KUKA KRL program: MyProgram_292().src

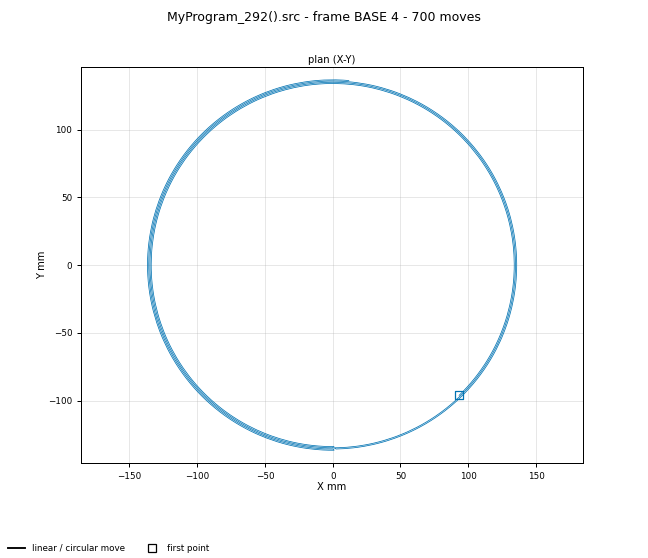
[picture p0: tool path of MyProgram_292().src in frame BASE 4, 700 of 700 moves have a stored position in this frame; points joined in program order, loops and branches not executed]
&ACCESS RVP
&REL 1
&PARAM TEMPLATE = C:\KRC\Roboter\Template\vorgabe
&PARAM EDITMASK = *
DEF MyProgram_292()
; ---- Setting reference (Base) ----
$BASE = BASE_DATA[4]

; --------------------------
; ---- Setting tool (TCP) ----
$TOOL = TOOL_DATA[3]
; --------------------------

$VEL.CP = VEL_APROX_PRINT
Startdeposition()
$VEL.CP = VEL_PRINT
LIN {X 93.2547,Y -96.1677,Z 177,A -42.5011,B 6.5222,C 0.3337,E1 6.6439,E2 494.4395} C_DIS
LIN {X 96.4506,Y -92.9625,Z 177,A -40.616,B 6.5225,C 0.3304,E1 6.6475,E2 492.5591} C_DIS
LIN {X 99.1155,Y -90.1154,Z 177,A -39.0001,B 6.5225,C 0.3277,E1 6.6506,E2 490.9482} C_DIS
LIN {X 101.7886,Y -87.0857,Z 177,A -37.2313,B 6.5228,C 0.3231,E1 6.6538,E2 489.1727} C_DIS
LIN {X 104.4652,Y -83.8557,Z 177,A -35.5009,B 6.523,C 0.3201,E1 6.6569,E2 487.4487} C_DIS
LIN {X 106.9431,Y -80.6711,Z 177,A -33.7806,B 6.5232,C 0.3162,E1 6.6598,E2 485.7275} C_DIS
LIN {X 109.619,Y -76.9961,Z 177,A -31.8796,B 6.5233,C 0.3123,E1 6.6629,E2 483.8301} C_DIS
LIN {X 112.1141,Y -73.3161,Z 177,A -30.1093,B 6.5235,C 0.3099,E1 6.6656,E2 482.0746} C_DIS
LIN {X 113.9637,Y -70.4067,Z 177,A -28.5276,B 6.5237,C 0.3044,E1 6.668,E2 480.478} C_DIS
LIN {X 115.9303,Y -67.118,Z 177,A -27.0187,B 6.5238,C 0.3025,E1 6.6701,E2 478.9839} C_DIS
LIN {X 118.1011,Y -63.2205,Z 177,A -25.0687,B 6.5241,C 0.2969,E1 6.6727,E2 477.0268} C_DIS
LIN {X 119.8057,Y -59.9271,Z 177,A -23.4735,B 6.5242,C 0.2926,E1 6.6747,E2 475.429} C_DIS
LIN {X 121.6866,Y -56.0049,Z 177,A -21.7807,B 6.5243,C 0.2906,E1 6.6767,E2 473.7555} C_DIS
LIN {X 122.9604,Y -53.1495,Z 177,A -20.5105,B 6.5244,C 0.2882,E1 6.6781,E2 472.4924} C_DIS
LIN {X 124.4377,Y -49.5951,Z 177,A -18.8101,B 6.5247,C 0.2828,E1 6.6799,E2 470.7838} C_DIS
LIN {X 125.9052,Y -45.7399,Z 177,A -17.0927,B 6.5248,C 0.2789,E1 6.6816,E2 469.0705} C_DIS
LIN {X 127.2852,Y -41.7458,Z 177,A -15.2801,B 6.5251,C 0.2738,E1 6.6832,E2 467.2556} C_DIS
LIN {X 128.7083,Y -37.1294,Z 177,A -12.2803,B 6.5259,C 0.2519,E1 6.6857,E2 464.1364} C_DIS
LIN {X 130.5683,Y -29.9352,Z 177,A -10.1949,B 6.5255,C 0.262,E1 6.6869,E2 462.1858} C_DIS
LIN {X 131.2974,Y -26.5557,Z 177,A -8.8361,B 6.5256,C 0.2599,E1 6.6877,E2 460.8406} C_DIS
LIN {X 131.8472,Y -23.6754,Z 177,A -7.5979,B 6.5258,C 0.2566,E1 6.6883,E2 459.6033} C_DIS
LIN {X 132.417,Y -20.2488,Z 177,A -6.0396,B 6.526,C 0.2511,E1 6.689,E2 458.0347} C_DIS
LIN {X 132.9133,Y -16.6972,Z 177,A -4.5118,B 6.5261,C 0.2469,E1 6.6895,E2 456.5064} C_DIS
LIN {X 133.3452,Y -12.7791,Z 177,A -2.9752,B 6.5262,C 0.2446,E1 6.69,E2 454.9869} C_DIS
LIN {X 133.6654,Y -8.842,Z 177,A -1.0029,B 6.5266,C 0.2349,E1 6.6904,E2 452.978} C_DIS
LIN {X 133.8408,Y -5.5702,Z 177,A -0.0788,B 6.5264,C 0.2391,E1 6.6904,E2 452.112} C_DIS
LIN {X 133.9241,Y -3.0185,Z 177,A 1.1002,B 6.5266,C 0.2345,E1 6.6906,E2 450.9214} C_DIS
LIN {X 133.9546,Y 0.822,Z 177,A 2.8788,B 6.5268,C 0.2274,E1 6.6906,E2 449.1246} C_DIS
LIN {X 133.879,Y 4.576,Z 177,A 4.2711,B 6.5268,C 0.2265,E1 6.6905,E2 447.7575} C_DIS
LIN {X 133.7434,Y 7.5752,Z 177,A 5.4943,B 6.527,C 0.2239,E1 6.6903,E2 446.5409} C_DIS
LIN {X 133.4661,Y 11.4487,Z 177,A 7.1189,B 6.527,C 0.2198,E1 6.6899,E2 444.9194} C_DIS
LIN {X 133.2196,Y 14.0308,Z 177,A 8.1651,B 6.5272,C 0.2177,E1 6.6897,E2 443.8802} C_DIS
LIN {X 132.9288,Y 16.5728,Z 177,A 9.3123,B 6.5272,C 0.2137,E1 6.6893,E2 442.7257} C_DIS
LIN {X 132.5516,Y 19.3507,Z 177,A 10.6317,B 6.5275,C 0.2082,E1 6.6887,E2 441.3905} C_DIS
LIN {X 131.8477,Y 23.6726,Z 177,A 12.355,B 6.5275,C 0.2055,E1 6.6879,E2 439.6844} C_DIS
LIN {X 131.2568,Y 26.7556,Z 177,A 13.6501,B 6.5277,C 0.2026,E1 6.6872,E2 438.3942} C_DIS
LIN {X 130.5423,Y 30.0492,Z 177,A 15.1238,B 6.5277,C 0.198,E1 6.6863,E2 436.9154} C_DIS
LIN {X 129.489,Y 34.3048,Z 177,A 16.9836,B 6.5279,C 0.1931,E1 6.685,E2 435.0563} C_DIS
LIN {X 128.2952,Y 38.5354,Z 177,A 19.333,B 6.5283,C 0.1799,E1 6.6831,E2 432.6477} C_DIS
LIN {X 126.8174,Y 43.1518,Z 177,A 20.7515,B 6.5282,C 0.1854,E1 6.682,E2 431.3088} C_DIS
LIN {X 124.899,Y 48.419,Z 177,A 23.6983,B 6.5286,C 0.1697,E1 6.679,E2 428.2928} C_DIS
LIN {X 123.0953,Y 52.8375,Z 177,A 24.9449,B 6.5284,C 0.1778,E1 6.6777,E2 427.1429} C_DIS
LIN {X 121.1405,Y 57.1795,Z 177,A 27.275,B 6.5286,C 0.1676,E1 6.675,E2 424.7758} C_DIS
LIN {X 119.2439,Y 61.0336,Z 177,A 28.926,B 6.5286,C 0.166,E1 6.6729,E2 423.1466} C_DIS
LIN {X 117.5054,Y 64.3209,Z 177,A 30.6108,B 6.5288,C 0.1604,E1 6.6707,E2 421.4496} C_DIS
LIN {X 115.2166,Y 68.3366,Z 177,A 32.5475,B 6.5289,C 0.1562,E1 6.668,E2 419.517} C_DIS
LIN {X 112.8881,Y 72.1176,Z 177,A 34.404,B 6.529,C 0.1523,E1 6.6652,E2 417.6649} C_DIS
LIN {X 110.2862,Y 76.0374,Z 177,A 36.2624,B 6.529,C 0.1501,E1 6.6623,E2 415.8244} C_DIS
LIN {X 107.7865,Y 79.5413,Z 177,A 38.1742,B 6.5292,C 0.1447,E1 6.6592,E2 413.9033} C_DIS
LIN {X 101.9515,Y 86.8941,Z 177,A 42.0062,B 6.5293,C 0.1388,E1 6.6525,E2 410.0924} C_DIS
LIN {X 99.4872,Y 89.7057,Z 177,A 43.7299,B 6.5294,C 0.1333,E1 6.6493,E2 408.353} C_DIS
LIN {X 96.1576,Y 93.2651,Z 177,A 45.6306,B 6.5294,C 0.132,E1 6.6457,E2 406.4741} C_DIS
LIN {X 93.4408,Y 95.9875,Z 177,A 47.3771,B 6.5295,C 0.127,E1 6.6422,E2 404.7149} C_DIS
LIN {X 90.2793,Y 98.9668,Z 177,A 49.225,B 6.5296,C 0.1236,E1 6.6384,E2 402.8678} C_DIS
LIN {X 87.6848,Y 101.2726,Z 177,A 50.6916,B 6.5296,C 0.1211,E1 6.6353,E2 401.4032} C_DIS
LIN {X 84.3245,Y 104.0871,Z 177,A 52.5309,B 6.5297,C 0.1182,E1 6.6313,E2 399.5678} C_DIS
LIN {X 80.8508,Y 106.8075,Z 177,A 54.3017,B 6.5297,C 0.1168,E1 6.6275,E2 397.8109} C_DIS
LIN {X 77.4949,Y 109.267,Z 177,A 56.7417,B 6.53,C 0.1034,E1 6.6217,E2 395.2904} C_DIS
LIN {X 72.9543,Y 112.3491,Z 177,A 58.2306,B 6.5298,C 0.1131,E1 6.6185,E2 393.9056} C_DIS
LIN {X 70.2551,Y 114.0567,Z 177,A 59.8013,B 6.5298,C 0.1079,E1 6.6147,E2 392.3102} C_DIS
LIN {X 67.1093,Y 115.9354,Z 177,A 61.3332,B 6.5299,C 0.1061,E1 6.611,E2 390.7826} C_DIS
LIN {X 63.6933,Y 117.8471,Z 177,A 63.0269,B 6.5299,C 0.1035,E1 6.6069,E2 389.0865} C_DIS
LIN {X 59.6278,Y 119.9533,Z 177,A 64.965,B 6.5299,C 0.1013,E1 6.602,E2 387.1509} C_DIS
LIN {X 55.7819,Y 121.7897,Z 177,A 66.6368,B 6.5299,C 0.1013,E1 6.5979,E2 385.4974} C_DIS
LIN {X 52.4854,Y 123.2475,Z 177,A 68.1681,B 6.53,C 0.0997,E1 6.5939,E2 383.9676} C_DIS
LIN {X 49.6492,Y 124.4159,Z 177,A 69.4709,B 6.53,C 0.0984,E1 6.5906,E2 382.666} C_DIS
LIN {X 45.9682,Y 125.8229,Z 177,A 71.4893,B 6.5301,C 0.0918,E1 6.5852,E2 380.6076} C_DIS
LIN {X 42.6946,Y 126.9704,Z 177,A 72.6051,B 6.5301,C 0.0958,E1 6.5824,E2 379.5365} C_DIS
LIN {X 35.9258,Y 129.0486,Z 177,A 75.9572,B 6.5301,C 0.0886,E1 6.5733,E2 376.1461} C_DIS
LIN {X 32.5628,Y 129.9385,Z 177,A 77.0114,B 6.5301,C 0.0938,E1 6.5706,E2 375.1444} C_DIS
LIN {X 29.6776,Y 130.6272,Z 177,A 78.365,B 6.5301,C 0.0917,E1 6.5669,E2 373.781} C_DIS
LIN {X 26.4894,Y 131.3109,Z 177,A 79.7722,B 6.5301,C 0.0907,E1 6.563,E2 372.3726} C_DIS
LIN {X 22.8852,Y 131.9886,Z 177,A 81.2873,B 6.5301,C 0.0907,E1 6.5589,E2 370.8645} C_DIS
LIN {X 19.5056,Y 132.5295,Z 177,A 82.849,B 6.5301,C 0.0886,E1 6.5545,E2 369.2915} C_DIS
LIN {X 15.2294,Y 133.0891,Z 177,A 84.594,B 6.5301,C 0.0894,E1 6.5497,E2 367.5591} C_DIS
LIN {X 11.0703,Y 133.4981,Z 177,A 86.315,B 6.5301,C 0.0898,E1 6.545,E2 365.8467} C_DIS
LIN {X 8.5569,Y 133.683,Z 177,A 87.5726,B 6.5302,C 0.0871,E1 6.5414,E2 364.568} C_DIS
LIN {X 4.6226,Y 133.8778,Z 177,A 89.1069,B 6.5302,C 0.0889,E1 6.5372,E2 363.0525} C_DIS
LIN {X 1.7234,Y 133.9461,Z 177,A 90.568,B 6.5302,C 0.0858,E1 6.533,E2 361.5654} C_DIS
LIN {X -2.809,Y 133.9281,Z 177,A 92.3744,B 6.5302,C 0.0876,E1 6.528,E2 359.7758} C_DIS
LIN {X -6.0372,Y 133.8219,Z 177,A 93.7882,B 6.5302,C 0.0873,E1 6.524,E2 358.3588} C_DIS
LIN {X -9.8651,Y 133.5924,Z 177,A 95.4536,B 6.5302,C 0.0873,E1 6.5194,E2 356.6912} C_DIS
LIN {X -14.4166,Y 133.1781,Z 177,A 97.3355,B 6.5302,C 0.0888,E1 6.5142,E2 354.819} C_DIS
LIN {X -17.6905,Y 132.7831,Z 177,A 98.7772,B 6.5302,C 0.0888,E1 6.5102,E2 353.3743} C_DIS
LIN {X -21.9534,Y 132.1449,Z 177,A 100.6192,B 6.5302,C 0.0897,E1 6.5051,E2 351.5336} C_DIS
LIN {X -25.4976,Y 131.5074,Z 177,A 102.0736,B 6.5302,C 0.0916,E1 6.5012,E2 350.0903} C_DIS
LIN {X -28.3851,Y 130.9141,Z 177,A 103.3903,B 6.5302,C 0.0916,E1 6.4975,E2 348.7677} C_DIS
LIN {X -32.2156,Y 130.0266,Z 177,A 105.0573,B 6.5302,C 0.0929,E1 6.493,E2 347.1036} C_DIS
LIN {X -34.716,Y 129.3794,Z 177,A 106.2071,B 6.5302,C 0.0931,E1 6.4899,E2 345.949} C_DIS
LIN {X -40.4025,Y 127.7182,Z 177,A 108.5712,B 6.5301,C 0.0973,E1 6.4836,E2 343.607} C_DIS
LIN {X -44.6966,Y 126.2813,Z 177,A 111.3947,B 6.5301,C 0.0878,E1 6.4759,E2 340.6783} C_DIS
LIN {X -49.5868,Y 124.441,Z 177,A 112.8347,B 6.5301,C 0.1001,E1 6.4724,E2 339.3355} C_DIS
LIN {X -51.7604,Y 123.5517,Z 177,A 114.0213,B 6.5301,C 0.0989,E1 6.4693,E2 338.1279} C_DIS
LIN {X -55.3587,Y 121.9839,Z 177,A 115.6589,B 6.53,C 0.1014,E1 6.4651,E2 336.4965} C_DIS
LIN {X -58.1429,Y 120.6802,Z 177,A 117.1082,B 6.53,C 0.1014,E1 6.4614,E2 335.032} C_DIS
LIN {X -61.7821,Y 118.8587,Z 177,A 119.1939,B 6.53,C 0.0994,E1 6.4562,E2 332.9061} C_DIS
LIN {X -65.3727,Y 116.9237,Z 177,A 120.3017,B 6.5299,C 0.1096,E1 6.4537,E2 331.8762} C_DIS
LIN {X -67.9903,Y 115.421,Z 177,A 121.9186,B 6.5299,C 0.1075,E1 6.4496,E2 330.2213} C_DIS
LIN {X -71.3651,Y 113.3653,Z 177,A 123.619,B 6.5299,C 0.1099,E1 6.4456,E2 328.5211} C_DIS
LIN {X -76.8897,Y 109.694,Z 177,A 126.2273,B 6.5297,C 0.1171,E1 6.4397,E2 325.9426} C_DIS
LIN {X -79.3379,Y 107.9359,Z 177,A 127.799,B 6.5297,C 0.1159,E1 6.436,E2 324.3381} C_DIS
LIN {X -82.8055,Y 105.2991,Z 177,A 129.6731,B 6.5297,C 0.1191,E1 6.4319,E2 322.4643} C_DIS
LIN {X -86.1951,Y 102.5431,Z 177,A 131.5799,B 6.5297,C 0.122,E1 6.4278,E2 320.5545} C_DIS
LIN {X -89.4519,Y 99.7147,Z 177,A 133.4568,B 6.5296,C 0.1252,E1 6.4238,E2 318.6753} C_DIS
LIN {X -92.8056,Y 96.6017,Z 177,A 135.4367,B 6.5296,C 0.1287,E1 6.4198,E2 316.6944} C_DIS
LIN {X -95.7212,Y 93.7129,Z 177,A 137.2067,B 6.5294,C 0.1321,E1 6.4163,E2 314.9243} C_DIS
LIN {X -98.7785,Y 90.4849,Z 177,A 139.1704,B 6.5294,C 0.1354,E1 6.4126,E2 312.9547} C_DIS
LIN {X -101.7402,Y 87.142,Z 177,A 141.1279,B 6.5294,C 0.139,E1 6.409,E2 310.9933} C_DIS
LIN {X -104.577,Y 83.7165,Z 177,A 143.05,B 6.5292,C 0.143,E1 6.4056,E2 309.0706} C_DIS
LIN {X -107.1431,Y 80.4061,Z 177,A 144.7491,B 6.5292,C 0.1482,E1 6.4027,E2 307.3842} C_DIS
LIN {X -109.243,Y 77.5291,Z 177,A 146.4559,B 6.5291,C 0.1497,E1 6.3999,E2 305.6568} C_DIS
LIN {X -112.9435,Y 72.0311,Z 177,A 149.2423,B 6.5289,C 0.157,E1 6.3956,E2 302.8788} C_DIS
LIN {X -115.0741,Y 68.5756,Z 177,A 151.0676,B 6.5289,C 0.1603,E1 6.393,E2 301.0444} C_DIS
LIN {X -116.8004,Y 65.5922,Z 177,A 152.5887,B 6.5287,C 0.1634,E1 6.3909,E2 299.519} C_DIS
LIN {X -118.933,Y 61.6406,Z 177,A 154.4238,B 6.5286,C 0.1692,E1 6.3885,E2 297.6959} C_DIS
LIN {X -120.4075,Y 58.7071,Z 177,A 155.9944,B 6.5286,C 0.171,E1 6.3865,E2 296.1066} C_DIS
LIN {X -123.0186,Y 53.015,Z 177,A 158.6392,B 6.5284,C 0.1784,E1 6.3835,E2 293.4683} C_DIS
LIN {X -124.3654,Y 49.7743,Z 177,A 160.1661,B 6.5283,C 0.1821,E1 6.3819,E2 291.9397} C_DIS
LIN {X -125.8482,Y 45.8979,Z 177,A 161.8282,B 6.5281,C 0.1881,E1 6.3803,E2 290.2929} C_DIS
LIN {X -126.6044,Y 43.7664,Z 177,A 163.0259,B 6.5281,C 0.1883,E1 6.3792,E2 289.0681} C_DIS
LIN {X -127.7431,Y 40.3247,Z 177,A 164.4677,B 6.5279,C 0.1937,E1 6.3779,E2 287.641} C_DIS
LIN {X -128.7727,Y 36.9097,Z 177,A 166.0775,B 6.5279,C 0.197,E1 6.3767,E2 286.0223} C_DIS
LIN {X -129.7111,Y 33.4588,Z 177,A 167.5354,B 6.5277,C 0.202,E1 6.3756,E2 284.5745} C_DIS
LIN {X -130.611,Y 29.7484,Z 177,A 169.3185,B 6.5276,C 0.2049,E1 6.3745,E2 282.7746} C_DIS
LIN {X -131.3492,Y 26.3015,Z 177,A 171.0086,B 6.5276,C 0.2072,E1 6.3735,E2 281.0637} C_DIS
LIN {X -132.1843,Y 21.7173,Z 177,A 172.9941,B 6.5273,C 0.2129,E1 6.3725,E2 279.0809} C_DIS
LIN {X -132.7482,Y 17.957,Z 177,A 174.509,B 6.5271,C 0.2188,E1 6.3719,E2 277.581} C_DIS
LIN {X -133.1057,Y 15.0892,Z 177,A 175.8069,B 6.5271,C 0.2216,E1 6.3715,E2 276.2767} C_DIS
LIN {X -133.4911,Y 11.1532,Z 177,A 177.5894,B 6.5269,C 0.2255,E1 6.3711,E2 274.4844} C_DIS
LIN {X -133.771,Y 7.049,Z 177,A 179.4151,B 6.5268,C 0.2298,E1 6.3708,E2 272.6522} C_DIS
LIN {X -133.9146,Y 3.3582,Z 177,A -179.067,B 6.5266,C 0.235,E1 6.3706,E2 271.1432} C_DIS
LIN {X -133.9568,Y 0.5032,Z 177,A -177.7907,B 6.5265,C 0.2379,E1 6.3706,E2 269.8612} C_DIS
LIN {X -133.9184,Y -3.2227,Z 177,A -176.0516,B 6.5264,C 0.2409,E1 6.3706,E2 268.1055} C_DIS
LIN {X -133.7767,Y -6.9356,Z 177,A -174.5652,B 6.5261,C 0.2465,E1 6.3709,E2 266.6329} C_DIS
LIN {X -133.5934,Y -9.8526,Z 177,A -173.2029,B 6.5261,C 0.2489,E1 6.3711,E2 265.2578} C_DIS
LIN {X -133.2061,Y -14.1561,Z 177,A -171.2366,B 6.5259,C 0.2528,E1 6.3717,E2 263.2785} C_DIS
LIN {X -132.6335,Y -18.7776,Z 177,A -169.2218,B 6.5257,C 0.2582,E1 6.3724,E2 261.2624} C_DIS
LIN {X -132.1135,Y -22.1417,Z 177,A -167.8158,B 6.5255,C 0.2629,E1 6.373,E2 259.8636} C_DIS
LIN {X -131.4967,Y -25.5535,Z 177,A -166.373,B 6.5253,C 0.2675,E1 6.3738,E2 258.4268} C_DIS
LIN {X -130.815,Y -28.8441,Z 177,A -164.5422,B 6.5253,C 0.2672,E1 6.3749,E2 256.5485} C_DIS
LIN {X -128.9504,Y -36.2767,Z 177,A -161.3851,B 6.5249,C 0.2775,E1 6.3771,E2 253.4086} C_DIS
LIN {X -127.969,Y -39.6012,Z 177,A -159.8428,B 6.5248,C 0.2809,E1 6.3784,E2 251.8598} C_DIS
LIN {X -126.8559,Y -43.0385,Z 177,A -158.4005,B 6.5245,C 0.2862,E1 6.3796,E2 250.4313} C_DIS
LIN {X -125.6963,Y -46.3153,Z 177,A -156.9142,B 6.5244,C 0.2902,E1 6.381,E2 248.9459} C_DIS
LIN {X -124.7138,Y -48.8954,Z 177,A -155.6899,B 6.5242,C 0.2928,E1 6.3823,E2 247.7169} C_DIS
LIN {X -123.2773,Y -52.4166,Z 177,A -154.0105,B 6.5241,C 0.2965,E1 6.3841,E2 246.032} C_DIS
LIN {X -121.9963,Y -55.331,Z 177,A -152.618,B 6.5239,C 0.2996,E1 6.3857,E2 244.6364} C_DIS
LIN {X -120.0449,Y -59.4422,Z 177,A -150.5894,B 6.5237,C 0.3036,E1 6.3881,E2 242.5986} C_DIS
LIN {X -118.4513,Y -62.5579,Z 177,A -148.1294,B 6.5241,C 0.2964,E1 6.3915,E2 240.0192} C_DIS
LIN {X -115.1617,Y -68.4287,Z 177,A -146.0824,B 6.5233,C 0.313,E1 6.3942,E2 238.0777} C_DIS
LIN {X -112.864,Y -72.1553,Z 177,A -144.1833,B 6.5231,C 0.3171,E1 6.3971,E2 236.1762} C_DIS
LIN {X -110.4263,Y -75.8333,Z 177,A -142.2092,B 6.5229,C 0.3205,E1 6.4002,E2 234.1921} C_DIS
LIN {X -107.7448,Y -79.598,Z 177,A -140.4774,B 6.5226,C 0.3278,E1 6.4029,E2 232.4915} C_DIS
LIN {X -106.0986,Y -81.7795,Z 177,A -138.87,B 6.5227,C 0.3253,E1 6.4058,E2 230.8299} C_DIS
LIN {X -103.506,Y -85.0369,Z 177,A -137.1986,B 6.5225,C 0.3304,E1 6.4087,E2 229.1728} C_DIS
LIN {X -100.6101,Y -88.4444,Z 177,A -135.2447,B 6.5223,C 0.3339,E1 6.4123,E2 227.2144} C_DIS
LIN {X -98.2184,Y -91.0927,Z 177,A -133.758,B 6.5221,C 0.3375,E1 6.4151,E2 225.733} C_DIS
LIN {X -95.549,Y -93.8885,Z 177,A -132.0971,B 6.5219,C 0.3407,E1 6.4183,E2 224.0716} C_DIS
LIN {X -92.7691,Y -96.6366,Z 177,A -130.3072,B 6.5219,C 0.3425,E1 6.4219,E2 222.2674} C_DIS
LIN {X -89.5256,Y -99.6487,Z 177,A -128.4052,B 6.5217,C 0.3459,E1 6.4258,E2 220.3647} C_DIS
LIN {X -86.0607,Y -102.6558,Z 177,A -126.4402,B 6.5215,C 0.3494,E1 6.43,E2 218.3997} C_DIS
LIN {X -82.3757,Y -105.6364,Z 177,A -124.476,B 6.5212,C 0.3536,E1 6.4343,E2 216.4437} C_DIS
LIN {X -79.5559,Y -107.7757,Z 177,A -122.4217,B 6.5215,C 0.3493,E1 6.4391,E2 214.3217} C_DIS
LIN {X -75.9885,Y -110.3198,Z 177,A -121.1933,B 6.5209,C 0.3603,E1 6.4417,E2 213.1745} C_DIS
LIN {X -73.3161,Y -112.1141,Z 177,A -119.5903,B 6.5209,C 0.3595,E1 6.4455,E2 211.5434} C_DIS
LIN {X -69.7205,Y -114.3847,Z 177,A -117.679,B 6.5209,C 0.3609,E1 6.45,E2 209.6205} C_DIS
LIN {X -66.3323,Y -116.3817,Z 177,A -116.0487,B 6.5207,C 0.3638,E1 6.454,E2 207.9967} C_DIS
LIN {X -62.6117,Y -118.4231,Z 177,A -114.1444,B 6.5207,C 0.3649,E1 6.4587,E2 206.0811} C_DIS
LIN {X -58.7482,Y -120.3873,Z 177,A -112.4268,B 6.5204,C 0.3689,E1 6.4629,E2 204.3806} C_DIS
LIN {X -56.2707,Y -121.5637,Z 177,A -111.2394,B 6.5204,C 0.37,E1 6.4659,E2 203.1912} C_DIS
LIN {X -52.6057,Y -123.1955,Z 177,A -109.4964,B 6.5203,C 0.3714,E1 6.4704,E2 201.4448} C_DIS
LIN {X -50.1212,Y -124.2256,Z 177,A -108.3301,B 6.5203,C 0.3723,E1 6.4734,E2 200.2762} C_DIS
LIN {X -45.5141,Y -125.9866,Z 177,A -106.3135,B 6.52,C 0.3755,E1 6.4787,E2 198.271} C_DIS
LIN {X -39.0025,Y -128.1523,Z 177,A -102.9244,B 6.5202,C 0.3716,E1 6.4878,E2 194.8242} C_DIS
LIN {X -35.6668,Y -129.121,Z 177,A -101.8519,B 6.5199,C 0.3782,E1 6.4906,E2 193.8036} C_DIS
LIN {X -32.7186,Y -129.8989,Z 177,A -100.476,B 6.5199,C 0.378,E1 6.4943,E2 192.4183} C_DIS
LIN {X -29.396,Y -130.6915,Z 177,A -98.9977,B 6.5199,C 0.3786,E1 6.4984,E2 190.9375} C_DIS
LIN {X -26.0141,Y -131.4077,Z 177,A -97.3468,B 6.5199,C 0.3769,E1 6.5029,E2 189.2645} C_DIS
LIN {X -21.9874,Y -132.1392,Z 177,A -95.6946,B 6.5199,C 0.3789,E1 6.5074,E2 187.624} C_DIS
LIN {X -18.1984,Y -132.7163,Z 177,A -94.1313,B 6.5197,C 0.3804,E1 6.5117,E2 186.0698} C_DIS
LIN {X -14.1879,Y -133.2027,Z 177,A -92.2621,B 6.5198,C 0.3788,E1 6.517,E2 184.182} C_DIS
LIN {X -10.5884,Y -133.5388,Z 177,A -90.8598,B 6.5198,C 0.381,E1 6.5208,E2 182.7973} C_DIS
LIN {X -6.8406,Y -133.7815,Z 177,A -89.1543,B 6.5198,C 0.3797,E1 6.5256,E2 181.0787} C_DIS
LIN {X -2.7749,Y -133.9286,Z 177,A -87.4107,B 6.5198,C 0.3795,E1 6.5305,E2 179.3339} C_DIS
LIN {X 0.9684,Y -133.9528,Z 177,A -86.2768,B 6.5194,C 0.3861,E1 6.5335,E2 178.258} C_DIS
Enddeposition()
LIN {X 0.9684,Y -133.9528,Z 177,A -86.2768,B 6.5194,C 0.3861,E1 6.5335,E2 178.258} C_DIS
Startdeposition()
$VEL.CP = VEL_PRINT
LIN {X -0.1253,Y -134.8623,Z 177,A -87.3645,B 6.5183,C 0.3988,E1 6.5298,E2 179.4573} C_DIS
LIN {X -3.8984,Y -134.8047,Z 177,A -88.8873,B 6.5183,C 0.3977,E1 6.5256,E2 180.9707} C_DIS
LIN {X -7.4524,Y -134.6566,Z 177,A -90.1989,B 6.5186,C 0.3949,E1 6.522,E2 182.258} C_DIS
LIN {X -11.2849,Y -134.388,Z 177,A -91.6976,B 6.5186,C 0.3928,E1 6.5179,E2 183.7406} C_DIS
LIN {X -18.9352,Y -133.525,Z 177,A -94.8815,B 6.5188,C 0.3909,E1 6.5091,E2 186.9148} C_DIS
LIN {X -22.0313,Y -133.0492,Z 177,A -96.3146,B 6.5188,C 0.3919,E1 6.5051,E2 188.3612} C_DIS
LIN {X -25.6748,Y -132.3947,Z 177,A -98.002,B 6.5187,C 0.3928,E1 6.5004,E2 190.0635} C_DIS
LIN {X -29.7309,Y -131.5431,Z 177,A -99.6989,B 6.5187,C 0.3911,E1 6.4958,E2 191.7529} C_DIS
LIN {X -32.9181,Y -130.7818,Z 177,A -101.0206,B 6.5189,C 0.3893,E1 6.4922,E2 193.066} C_DIS
LIN {X -36.0986,Y -129.9397,Z 177,A -102.3929,B 6.5189,C 0.3881,E1 6.4886,E2 194.4356} C_DIS
LIN {X -38.4704,Y -129.2586,Z 177,A -103.5047,B 6.5189,C 0.3882,E1 6.4855,E2 195.5556} C_DIS
LIN {X -44.5061,Y -127.3056,Z 177,A -106.2679,B 6.519,C 0.387,E1 6.4782,E2 198.3279} C_DIS
LIN {X -48.2453,Y -125.9373,Z 177,A -107.8626,B 6.5192,C 0.3842,E1 6.4741,E2 199.9106} C_DIS
LIN {X -51.6391,Y -124.5828,Z 177,A -109.5405,B 6.5192,C 0.3844,E1 6.4697,E2 201.6044} C_DIS
LIN {X -54.7986,Y -123.2256,Z 177,A -110.9861,B 6.5192,C 0.3827,E1 6.466,E2 203.0483} C_DIS
LIN {X -57.9363,Y -121.7816,Z 177,A -112.5318,B 6.5193,C 0.3821,E1 6.462,E2 204.6039} C_DIS
LIN {X -61.1039,Y -120.2234,Z 177,A -113.952,B 6.5195,C 0.3793,E1 6.4585,E2 206.0142} C_DIS
LIN {X -64.3645,Y -118.5122,Z 177,A -115.6527,B 6.5195,C 0.3791,E1 6.4543,E2 207.7321} C_DIS
LIN {X -68.2558,Y -116.3144,Z 177,A -117.5419,B 6.5196,C 0.3764,E1 6.4497,E2 209.6201} C_DIS
LIN {X -72.0083,Y -114.0293,Z 177,A -119.4512,B 6.5198,C 0.3743,E1 6.4452,E2 211.5346} C_DIS
LIN {X -75.8494,Y -111.5116,Z 177,A -121.169,B 6.5201,C 0.3685,E1 6.4412,E2 213.2232} C_DIS
LIN {X -79.536,Y -108.9124,Z 177,A -123.5047,B 6.52,C 0.3707,E1 6.4358,E2 215.611} C_DIS
LIN {X -83.7433,Y -105.7116,Z 177,A -125.6786,B 6.5202,C 0.366,E1 6.431,E2 217.7756} C_DIS
LIN {X -87.4973,Y -102.6262,Z 177,A -127.7456,B 6.5204,C 0.3624,E1 6.4266,E2 219.8426} C_DIS
LIN {X -90.8719,Y -99.6509,Z 177,A -129.6895,B 6.5206,C 0.3593,E1 6.4226,E2 221.7902} C_DIS
LIN {X -94.0855,Y -96.6227,Z 177,A -131.6015,B 6.5208,C 0.3562,E1 6.4187,E2 223.7062} C_DIS
LIN {X -97.0469,Y -93.6474,Z 177,A -133.3214,B 6.521,C 0.3519,E1 6.4153,E2 225.4178} C_DIS
LIN {X -99.005,Y -91.5755,Z 177,A -134.8011,B 6.521,C 0.3526,E1 6.4125,E2 226.9304} C_DIS
LIN {X -102.4643,Y -87.6877,Z 177,A -136.9033,B 6.5213,C 0.3467,E1 6.4086,E2 229.0185} C_DIS
LIN {X -105.6782,Y -83.7859,Z 177,A -139.5499,B 6.5213,C 0.3479,E1 6.4039,E2 231.7258} C_DIS
LIN {X -108.5854,Y -79.982,Z 177,A -140.9031,B 6.5219,C 0.3355,E1 6.4018,E2 232.9943} C_DIS
LIN {X -110.2852,Y -77.6213,Z 177,A -142.8241,B 6.5216,C 0.3405,E1 6.3986,E2 234.9993} C_DIS
LIN {X -112.8316,Y -73.8718,Z 177,A -144.294,B 6.5221,C 0.3308,E1 6.3964,E2 236.4124} C_DIS
LIN {X -115.0267,Y -70.4043,Z 177,A -146.0764,B 6.5223,C 0.3271,E1 6.3937,E2 238.1988} C_DIS
LIN {X -118.0456,Y -65.216,Z 177,A -149.1035,B 6.5223,C 0.3262,E1 6.3895,E2 241.2833} C_DIS
LIN {X -119.9785,Y -61.5849,Z 177,A -150.4338,B 6.5228,C 0.3172,E1 6.3879,E2 242.5615} C_DIS
LIN {X -121.4846,Y -58.5582,Z 177,A -152.0401,B 6.5228,C 0.3154,E1 6.3859,E2 244.1879} C_DIS
LIN {X -123.5502,Y -54.0652,Z 177,A -154.1328,B 6.5231,C 0.3099,E1 6.3835,E2 246.2784} C_DIS
LIN {X -125.0131,Y -50.5878,Z 177,A -155.6432,B 6.5234,C 0.3047,E1 6.3819,E2 247.7766} C_DIS
LIN {X -126.9204,Y -45.5918,Z 177,A -157.9289,B 6.5236,C 0.2988,E1 6.3796,E2 250.0626} C_DIS
LIN {X -127.8897,Y -42.7977,Z 177,A -159.2859,B 6.5237,C 0.2966,E1 6.3784,E2 251.4312} C_DIS
LIN {X -128.8416,Y -39.8419,Z 177,A -161.061,B 6.5237,C 0.298,E1 6.3769,E2 253.2611} C_DIS
LIN {X -129.9875,Y -35.9278,Z 177,A -161.9376,B 6.5243,C 0.2839,E1 6.3763,E2 254.0317} C_DIS
LIN {X -131.4598,Y -30.0952,Z 177,A -164.9497,B 6.5243,C 0.2819,E1 6.3742,E2 257.0984} C_DIS
LIN {X -132.1694,Y -26.808,Z 177,A -166.468,B 6.5245,C 0.2788,E1 6.3733,E2 258.6267} C_DIS
LIN {X -132.9616,Y -22.5559,Z 177,A -168.3487,B 6.5247,C 0.2741,E1 6.3724,E2 260.5113} C_DIS
LIN {X -133.576,Y -18.5784,Z 177,A -170.1782,B 6.5249,C 0.2706,E1 6.3717,E2 262.3542} C_DIS
LIN {X -134.089,Y -14.4084,Z 177,A -171.8696,B 6.5251,C 0.2645,E1 6.3711,E2 264.0329} C_DIS
LIN {X -134.3979,Y -11.1675,Z 177,A -173.3627,B 6.5252,C 0.2618,E1 6.3707,E2 265.5383} C_DIS
LIN {X -134.6773,Y -7.041,Z 177,A -175.1502,B 6.5254,C 0.2571,E1 6.3704,E2 267.3281} C_DIS
LIN {X -134.8247,Y -3.1804,Z 177,A -176.7847,B 6.5256,C 0.2523,E1 6.3703,E2 268.9605} C_DIS
LIN {X -134.8643,Y 0.1004,Z 177,A -178.3851,B 6.5256,C 0.2506,E1 6.3703,E2 270.585} C_DIS
LIN {X -134.7871,Y 4.5235,Z 177,A 179.7274,B 6.5259,C 0.2453,E1 6.3704,E2 272.4719} C_DIS
LIN {X -134.5783,Y 8.7378,Z 177,A 177.9383,B 6.5261,C 0.2401,E1 6.3707,E2 274.259} C_DIS
LIN {X -134.2499,Y 12.8226,Z 177,A 176.1701,B 6.5262,C 0.2354,E1 6.3711,E2 276.029} C_DIS
LIN {X -133.7905,Y 16.9664,Z 177,A 174.374,B 6.5264,C 0.2306,E1 6.3717,E2 277.8266} C_DIS
LIN {X -133.2476,Y 20.7974,Z 177,A 172.7283,B 6.5266,C 0.226,E1 6.3724,E2 279.471} C_DIS
LIN {X -132.5311,Y 24.9614,Z 177,A 170.8601,B 6.5267,C 0.2217,E1 6.3733,E2 281.3465} C_DIS
LIN {X -131.7898,Y 28.616,Z 177,A 169.2781,B 6.5269,C 0.2172,E1 6.3742,E2 282.9269} C_DIS
LIN {X -130.963,Y 32.1943,Z 177,A 167.7151,B 6.5269,C 0.2129,E1 6.3752,E2 284.4888} C_DIS
LIN {X -130.1284,Y 35.4184,Z 177,A 166.1433,B 6.5271,C 0.2107,E1 6.3764,E2 286.0784} C_DIS
LIN {X -129.1206,Y 38.9301,Z 177,A 164.6908,B 6.5272,C 0.2053,E1 6.3775,E2 287.5174} C_DIS
LIN {X -128.1439,Y 42.0344,Z 177,A 163.3201,B 6.5274,C 0.2014,E1 6.3787,E2 288.8854} C_DIS
LIN {X -127.4483,Y 44.0943,Z 177,A 161.8531,B 6.5273,C 0.2047,E1 6.3801,E2 290.4168} C_DIS
LIN {X -126.0121,Y 48.0514,Z 177,A 160.3252,B 6.5275,C 0.1971,E1 6.3816,E2 291.912} C_DIS
LIN {X -124.5495,Y 51.7188,Z 177,A 158.7781,B 6.5277,C 0.1913,E1 6.3832,E2 293.4418} C_DIS
LIN {X -123.1137,Y 55.0487,Z 177,A 157.0108,B 6.5277,C 0.1897,E1 6.3852,E2 295.2349} C_DIS
LIN {X -121.2164,Y 59.1126,Z 177,A 154.7498,B 6.5277,C 0.1886,E1 6.388,E2 297.5368} C_DIS
LIN {X -119.3107,Y 62.8676,Z 177,A 153.4375,B 6.528,C 0.1788,E1 6.3896,E2 298.7904} C_DIS
LIN {X -117.4227,Y 66.3315,Z 177,A 151.7013,B 6.5281,C 0.1753,E1 6.3919,E2 300.5323} C_DIS
LIN {X -115.7328,Y 69.2376,Z 177,A 150.2728,B 6.5282,C 0.1718,E1 6.394,E2 301.9595} C_DIS
LIN {X -113.2473,Y 73.2325,Z 177,A 147.9311,B 6.5282,C 0.1707,E1 6.3975,E2 304.3404} C_DIS
LIN {X -111.4588,Y 75.9274,Z 177,A 146.7016,B 6.5284,C 0.1658,E1 6.3994,E2 305.5514} C_DIS
LIN {X -108.9617,Y 79.4694,Z 177,A 144.818,B 6.5284,C 0.162,E1 6.4025,E2 307.4384} C_DIS
LIN {X -106.3105,Y 82.9827,Z 177,A 142.9003,B 6.5285,C 0.1583,E1 6.4058,E2 309.36} C_DIS
LIN {X -103.489,Y 86.4753,Z 177,A 140.9927,B 6.5286,C 0.1541,E1 6.4091,E2 311.266} C_DIS
LIN {X -100.5813,Y 89.8405,Z 177,A 139.0757,B 6.5287,C 0.1503,E1 6.4127,E2 313.1845} C_DIS
LIN {X -97.4754,Y 93.201,Z 177,A 137.1258,B 6.5288,C 0.1463,E1 6.4164,E2 315.1334} C_DIS
LIN {X -94.3207,Y 96.3924,Z 177,A 135.1771,B 6.5288,C 0.1429,E1 6.4203,E2 317.0854} C_DIS
LIN {X -90.9994,Y 99.5345,Z 177,A 133.1795,B 6.529,C 0.1398,E1 6.4244,E2 319.088} C_DIS
LIN {X -87.6576,Y 102.4899,Z 177,A 131.2277,B 6.529,C 0.1369,E1 6.4285,E2 321.0449} C_DIS
LIN {X -84.2297,Y 105.3249,Z 177,A 129.3657,B 6.5291,C 0.1331,E1 6.4325,E2 322.9019} C_DIS
LIN {X -80.8956,Y 107.9072,Z 177,A 127.5487,B 6.5291,C 0.1303,E1 6.4365,E2 324.7205} C_DIS
LIN {X -77.3733,Y 110.46,Z 177,A 125.7125,B 6.5292,C 0.1271,E1 6.4407,E2 326.5537} C_DIS
LIN {X -74.754,Y 112.2486,Z 177,A 123.6035,B 6.5291,C 0.134,E1 6.4459,E2 328.7517} C_DIS
LIN {X -69.8406,Y 115.3697,Z 177,A 121.6957,B 6.5293,C 0.1236,E1 6.4502,E2 330.5909} C_DIS
LIN {X -66.2706,Y 117.457,Z 177,A 119.2925,B 6.5292,C 0.1289,E1 6.4563,E2 333.069} C_DIS
LIN {X -61.0745,Y 120.2383,Z 177,A 117.5213,B 6.5294,C 0.1168,E1 6.4604,E2 334.7517} C_DIS
LIN {X -56.9868,Y 122.2294,Z 177,A 115.6229,B 6.5294,C 0.114,E1 6.4652,E2 336.6447} C_DIS
LIN {X -53.8734,Y 123.6331,Z 177,A 113.9484,B 6.5294,C 0.1151,E1 6.4695,E2 338.3447} C_DIS
LIN {X -49.6808,Y 125.3787,Z 177,A 111.3162,B 6.5294,C 0.1218,E1 6.4766,E2 341.0585} C_DIS
LIN {X -43.6793,Y 127.5922,Z 177,A 109.3587,B 6.5295,C 0.1098,E1 6.4815,E2 342.9246} C_DIS
LIN {X -39.0417,Y 129.0863,Z 177,A 107.0523,B 6.5295,C 0.111,E1 6.4877,E2 345.2576} C_DIS
LIN {X -35.5141,Y 130.1029,Z 177,A 105.7158,B 6.5295,C 0.107,E1 6.4912,E2 346.5667} C_DIS
LIN {X -31.9013,Y 131.0336,Z 177,A 104.2406,B 6.5296,C 0.1045,E1 6.4952,E2 348.0278} C_DIS
LIN {X -28.4768,Y 131.8199,Z 177,A 102.7039,B 6.5296,C 0.1042,E1 6.4994,E2 349.5687} C_DIS
LIN {X -24.2877,Y 132.6568,Z 177,A 100.8304,B 6.5296,C 0.104,E1 6.5046,E2 351.4482} C_DIS
LIN {X -20.5742,Y 133.2822,Z 177,A 99.3146,B 6.5296,C 0.1022,E1 6.5087,E2 352.953} C_DIS
LIN {X -16.9113,Y 133.7978,Z 177,A 97.6123,B 6.5296,C 0.1033,E1 6.5135,E2 354.6701} C_DIS
LIN {X -13.0866,Y 134.2246,Z 177,A 96.1109,B 6.5296,C 0.1011,E1 6.5176,E2 356.1547} C_DIS
LIN {X -8.3533,Y 134.602,Z 177,A 94.0559,B 6.5296,C 0.1012,E1 6.5233,E2 358.2132} C_DIS
LIN {X -4.5342,Y 134.7867,Z 177,A 92.402,B 6.5296,C 0.1015,E1 6.5279,E2 359.8699} C_DIS
LIN {X 0.2151,Y 134.8619,Z 177,A 90.1226,B 6.5296,C 0.105,E1 6.5344,E2 362.1794} C_DIS
LIN {X 3.4855,Y 134.8162,Z 177,A 88.9191,B 6.5296,C 0.1026,E1 6.5377,E2 363.3602} C_DIS
LIN {X 7.8399,Y 134.6336,Z 177,A 87.1211,B 6.5296,C 0.1021,E1 6.5427,E2 365.1511} C_DIS
LIN {X 10.7268,Y 134.4351,Z 177,A 85.4633,B 6.5296,C 0.1084,E1 6.5475,E2 366.8593} C_DIS
LIN {X 15.0794,Y 134.0168,Z 177,A 83.9936,B 6.5296,C 0.1036,E1 6.5514,E2 368.2824} C_DIS
LIN {X 19.4004,Y 133.4585,Z 177,A 82.1564,B 6.5296,C 0.1041,E1 6.5565,E2 370.1173} C_DIS
LIN {X 23.3237,Y 132.8293,Z 177,A 80.4812,B 6.5296,C 0.1048,E1 6.5611,E2 371.7904} C_DIS
LIN {X 27.4105,Y 132.0468,Z 177,A 78.7049,B 6.5296,C 0.1059,E1 6.5659,E2 373.5673} C_DIS
LIN {X 31.3332,Y 131.1705,Z 177,A 77.1277,B 6.5296,C 0.1052,E1 6.5702,E2 375.1284} C_DIS
LIN {X 34.3374,Y 130.4167,Z 177,A 75.9801,B 6.5296,C 0.1037,E1 6.5732,E2 376.2555} C_DIS
LIN {X 36.7834,Y 129.7478,Z 177,A 74.1459,B 6.5294,C 0.1155,E1 6.5784,E2 378.1797} C_DIS
LIN {X 41.4951,Y 128.319,Z 177,A 72.5368,B 6.5295,C 0.1104,E1 6.5825,E2 379.7311} C_DIS
LIN {X 45.5632,Y 126.9307,Z 177,A 70.7411,B 6.5295,C 0.1117,E1 6.5873,E2 381.5229} C_DIS
LIN {X 49.9502,Y 125.2701,Z 177,A 68.8288,B 6.5295,C 0.1125,E1 6.5922,E2 383.4253} C_DIS
LIN {X 53.3698,Y 123.8509,Z 177,A 67.3587,B 6.5295,C 0.1128,E1 6.596,E2 384.8829} C_DIS
LIN {X 56.56,Y 122.4267,Z 177,A 65.8713,B 6.5295,C 0.1146,E1 6.5998,E2 386.3705} C_DIS
LIN {X 59.5231,Y 121.0139,Z 177,A 64.5786,B 6.5295,C 0.1148,E1 6.603,E2 387.6509} C_DIS
LIN {X 62.484,Y 119.5121,Z 177,A 63.0537,B 6.5294,C 0.1184,E1 6.6068,E2 389.1895} C_DIS
LIN {X 66.0039,Y 117.6069,Z 177,A 61.3126,B 6.5294,C 0.1214,E1 6.6111,E2 390.9355} C_DIS
LIN {X 69.7475,Y 115.426,Z 177,A 59.5079,B 6.5293,C 0.1235,E1 6.6154,E2 392.736} C_DIS
LIN {X 73.352,Y 113.1697,Z 177,A 57.7856,B 6.5293,C 0.125,E1 6.6194,E2 394.4482} C_DIS
LIN {X 77.6757,Y 110.2468,Z 177,A 55.5047,B 6.5292,C 0.1296,E1 6.6247,E2 396.737} C_DIS
LIN {X 81.2953,Y 107.6056,Z 177,A 53.6328,B 6.5292,C 0.1324,E1 6.6289,E2 398.6053} C_DIS
LIN {X 84.8881,Y 104.7949,Z 177,A 51.725,B 6.5291,C 0.1354,E1 6.6331,E2 400.5098} C_DIS
LIN {X 88.3103,Y 101.9281,Z 177,A 49.8277,B 6.529,C 0.1389,E1 6.6371,E2 402.4075} C_DIS
LIN {X 92.854,Y 97.8069,Z 177,A 47.2476,B 6.5289,C 0.1435,E1 6.6424,E2 404.985} C_DIS
LIN {X 95.9918,Y 94.7292,Z 177,A 45.1207,B 6.5287,C 0.1515,E1 6.6467,E2 407.1436} C_DIS
LIN {X 98.672,Y 91.9332,Z 177,A 43.8555,B 6.5287,C 0.1488,E1 6.649,E2 408.3635} C_DIS
LIN {X 101.4753,Y 88.8296,Z 177,A 42.068,B 6.5287,C 0.1528,E1 6.6523,E2 410.1528} C_DIS
LIN {X 104.5837,Y 85.147,Z 177,A 39.6773,B 6.5284,C 0.1628,E1 6.6566,E2 412.5855} C_DIS
LIN {X 107.2456,Y 81.7697,Z 177,A 38.2656,B 6.5284,C 0.1602,E1 6.6589,E2 413.9479} C_DIS
LIN {X 109.6658,Y 78.4939,Z 177,A 36.606,B 6.5284,C 0.1631,E1 6.6617,E2 415.5996} C_DIS
LIN {X 112.0121,Y 75.1082,Z 177,A 34.8504,B 6.5284,C 0.1673,E1 6.6644,E2 417.3565} C_DIS
LIN {X 114.3852,Y 71.442,Z 177,A 33.0263,B 6.5282,C 0.1713,E1 6.6671,E2 419.1777} C_DIS
LIN {X 116.6802,Y 67.6285,Z 177,A 31.1823,B 6.5282,C 0.1751,E1 6.6698,E2 421.0168} C_DIS
LIN {X 118.8229,Y 63.7888,Z 177,A 29.3137,B 6.528,C 0.1798,E1 6.6723,E2 422.8863} C_DIS
LIN {X 120.7008,Y 60.1579,Z 177,A 27.7573,B 6.528,C 0.1812,E1 6.6742,E2 424.4216} C_DIS
LIN {X 122.2949,Y 56.8451,Z 177,A 26.3575,B 6.528,C 0.1825,E1 6.6759,E2 425.8025} C_DIS
LIN {X 123.628,Y 53.8852,Z 177,A 25.0135,B 6.5278,C 0.1856,E1 6.6774,E2 427.143} C_DIS
LIN {X 125.0084,Y 50.5993,Z 177,A 22.7812,B 6.5274,C 0.2016,E1 6.6799,E2 429.4635} C_DIS
LIN {X 126.7498,Y 46.0648,Z 177,A 21.3097,B 6.5274,C 0.1972,E1 6.6812,E2 430.8643} C_DIS
LIN {X 127.8895,Y 42.7984,Z 177,A 19.7894,B 6.5274,C 0.202,E1 6.6826,E2 432.3917} C_DIS
LIN {X 129.3231,Y 38.2498,Z 177,A 17.8832,B 6.5272,C 0.2055,E1 6.6841,E2 434.2845} C_DIS
LIN {X 130.3737,Y 34.4988,Z 177,A 16.2619,B 6.5272,C 0.2095,E1 6.6853,E2 435.9028} C_DIS
LIN {X 131.3953,Y 30.3777,Z 177,A 14.5454,B 6.527,C 0.213,E1 6.6864,E2 437.6099} C_DIS
LIN {X 132.0776,Y 27.2593,Z 177,A 13.1863,B 6.5269,C 0.2169,E1 6.6872,E2 438.9702} C_DIS
LIN {X 132.6983,Y 24.0558,Z 177,A 11.8299,B 6.5268,C 0.2203,E1 6.6879,E2 440.324} C_DIS
LIN {X 133.245,Y 20.8144,Z 177,A 10.4887,B 6.5267,C 0.2233,E1 6.6885,E2 441.6593} C_DIS
LIN {X 133.7165,Y 17.5312,Z 177,A 9.1709,B 6.5266,C 0.2257,E1 6.689,E2 442.9669} C_DIS
LIN {X 134.0956,Y 14.3465,Z 177,A 7.7501,B 6.5264,C 0.2306,E1 6.6895,E2 444.3959} C_DIS
LIN {X 134.452,Y 10.5181,Z 177,A 6.0949,B 6.5262,C 0.2356,E1 6.6899,E2 446.0551} C_DIS
LIN {X 134.7394,Y 5.7473,Z 177,A 3.9341,B 6.5259,C 0.2436,E1 6.6902,E2 448.2336} C_DIS
LIN {X 134.8645,Y 0.0714,Z 177,A 1.7016,B 6.5258,C 0.2475,E1 6.6902,E2 450.4459} C_DIS
LIN {X 134.7832,Y -4.6228,Z 177,A -0.8888,B 6.5252,C 0.2634,E1 6.69,E2 453.111} C_DIS
LIN {X 134.4568,Y -10.4515,Z 177,A -2.6212,B 6.5254,C 0.2577,E1 6.6897,E2 454.7537} C_DIS
LIN {X 134.0892,Y -14.4062,Z 177,A -4.1218,B 6.5254,C 0.2593,E1 6.6893,E2 456.2327} C_DIS
LIN {X 133.7267,Y -17.4532,Z 177,A -5.4521,B 6.5252,C 0.2635,E1 6.6888,E2 457.5673} C_DIS
LIN {X 133.2673,Y -20.6701,Z 177,A -6.8215,B 6.525,C 0.2672,E1 6.6883,E2 458.9365} C_DIS
LIN {X 132.829,Y -23.3252,Z 177,A -7.925,B 6.525,C 0.2698,E1 6.6878,E2 460.0361} C_DIS
LIN {X 132.1687,Y -26.8116,Z 177,A -9.4969,B 6.5247,C 0.2751,E1 6.6869,E2 461.6174} C_DIS
LIN {X 131.318,Y -30.716,Z 177,A -11.2234,B 6.5245,C 0.2804,E1 6.6858,E2 463.349} C_DIS
LIN {X 129.5755,Y -37.3878,Z 177,A -14.0359,B 6.5242,C 0.2866,E1 6.6838,E2 466.1496} C_DIS
LIN {X 128.5616,Y -40.7357,Z 177,A -15.2302,B 6.5242,C 0.2857,E1 6.6828,E2 467.309} C_DIS
LIN {X 127.0551,Y -45.218,Z 177,A -17.4294,B 6.5238,C 0.2944,E1 6.6808,E2 469.5337} C_DIS
LIN {X 125.0015,Y -50.6165,Z 177,A -19.8051,B 6.5236,C 0.2997,E1 6.6785,E2 471.9019} C_DIS
LIN {X 123.4789,Y -54.2302,Z 177,A -21.4797,B 6.5234,C 0.3043,E1 6.6766,E2 473.5793} C_DIS
LIN {X 121.8506,Y -57.792,Z 177,A -23.0688,B 6.5232,C 0.3074,E1 6.6747,E2 475.1605} C_DIS
LIN {X 120.4363,Y -60.6855,Z 177,A -24.2695,B 6.5232,C 0.3081,E1 6.6733,E2 476.3416} C_DIS
LIN {X 117.9763,Y -65.3412,Z 177,A -26.6576,B 6.5228,C 0.3164,E1 6.6701,E2 478.7507} C_DIS
LIN {X 115.9512,Y -68.8712,Z 177,A -28.3575,B 6.5226,C 0.3203,E1 6.6677,E2 480.4486} C_DIS
LIN {X 113.6148,Y -72.6606,Z 177,A -30.1563,B 6.5225,C 0.3234,E1 6.665,E2 482.2376} C_DIS
LIN {X 111.4181,Y -75.9871,Z 177,A -31.8964,B 6.5222,C 0.3283,E1 6.6623,E2 483.9851} C_DIS
LIN {X 108.8726,Y -79.5911,Z 177,A -33.7517,B 6.522,C 0.3325,E1 6.6593,E2 485.8398} C_DIS
LIN {X 106.0656,Y -83.2945,Z 177,A -35.6531,B 6.5219,C 0.3358,E1 6.6561,E2 487.7339} C_DIS
LIN {X 103.1623,Y -86.8646,Z 177,A -37.5671,B 6.5217,C 0.3396,E1 6.6527,E2 489.6446} C_DIS
LIN {X 100.267,Y -90.1914,Z 177,A -39.4236,B 6.5215,C 0.3435,E1 6.6492,E2 491.5006} C_DIS
LIN {X 97.2715,Y -93.4143,Z 177,A -41.2544,B 6.5213,C 0.3468,E1 6.6457,E2 493.3284} C_DIS
LIN {X 94.1722,Y -96.5381,Z 177,A -42.8467,B 6.5213,C 0.3462,E1 6.6427,E2 494.8875} C_DIS
LIN {X 90.2195,Y -100.2418,Z 177,A -45.3622,B 6.5209,C 0.3544,E1 6.6375,E2 497.432} C_DIS
LIN {X 86.9429,Y -103.0967,Z 177,A -47.2211,B 6.5207,C 0.3582,E1 6.6335,E2 499.2941} C_DIS
LIN {X 83.4089,Y -105.9757,Z 177,A -49.0942,B 6.5205,C 0.3607,E1 6.6294,E2 501.161} C_DIS
LIN {X 79.7533,Y -108.7534,Z 177,A -50.9701,B 6.5205,C 0.3631,E1 6.6252,E2 503.0292} C_DIS
LIN {X 76.2891,Y -111.2109,Z 177,A -52.7698,B 6.5202,C 0.3661,E1 6.6211,E2 504.8299} C_DIS
LIN {X 72.6115,Y -113.6462,Z 177,A -54.6484,B 6.5201,C 0.3693,E1 6.6167,E2 506.7106} C_DIS
LIN {X 68.771,Y -116.0109,Z 177,A -56.5376,B 6.5199,C 0.3719,E1 6.6122,E2 508.598} C_DIS
LIN {X 65.1469,Y -118.0839,Z 177,A -58.2234,B 6.5199,C 0.3731,E1 6.6081,E2 510.2742} C_DIS
LIN {X 61.8158,Y -119.8609,Z 177,A -59.7307,B 6.5198,C 0.3739,E1 6.6044,E2 511.7706} C_DIS
LIN {X 58.5906,Y -121.4691,Z 177,A -61.2405,B 6.5197,C 0.3757,E1 6.6007,E2 513.2789} C_DIS
LIN {X 55.6947,Y -122.8248,Z 177,A -62.6576,B 6.5195,C 0.3784,E1 6.597,E2 514.7044} C_DIS
LIN {X 52.5865,Y -124.1872,Z 177,A -64.7427,B 6.5188,C 0.3901,E1 6.5915,E2 516.8712} C_DIS
LIN {X 47.7139,Y -126.1386,Z 177,A -66.1396,B 6.5195,C 0.3798,E1 6.5881,E2 518.1653} C_DIS
LIN {X 44.6813,Y -127.2448,Z 177,A -68.0819,B 6.5188,C 0.39,E1 6.5828,E2 520.1804} C_DIS
LIN {X 40.8942,Y -128.5109,Z 177,A -69.3057,B 6.5192,C 0.3845,E1 6.5797,E2 521.346} C_DIS
LIN {X 38.0063,Y -129.3944,Z 177,A -70.5956,B 6.5191,C 0.3858,E1 6.5762,E2 522.6376} C_DIS
LIN {X 34.4894,Y -130.3762,Z 177,A -72.1678,B 6.5191,C 0.3875,E1 6.572,E2 524.2135} C_DIS
LIN {X 30.3777,Y -131.3953,Z 177,A -73.9352,B 6.5189,C 0.3884,E1 6.5672,E2 525.978} C_DIS
LIN {X 26.9562,Y -132.1393,Z 177,A -75.4038,B 6.5189,C 0.3892,E1 6.5632,E2 527.4452} C_DIS
LIN {X 23.6259,Y -132.7752,Z 177,A -77.0569,B 6.5187,C 0.3932,E1 6.5586,E2 529.1258} C_DIS
LIN {X 19.2989,Y -133.473,Z 177,A -78.6776,B 6.5188,C 0.3907,E1 6.5542,E2 530.7173} C_DIS
LIN {X 16.0003,Y -133.9083,Z 177,A -80.0986,B 6.5188,C 0.3915,E1 6.5502,E2 532.14} C_DIS
LIN {X 10.5635,Y -134.4487,Z 177,A -82.4483,B 6.5187,C 0.3928,E1 6.5437,E2 534.4947} C_DIS
LIN {X 4.2431,Y -134.7952,Z 177,A -85.0608,B 6.5187,C 0.3924,E1 6.5364,E2 537.0989} C_DIS
LIN {X 0.9725,Y -134.8573,Z 177,A -86.3065,B 6.5188,C 0.3905,E1 6.533,E2 538.3271} C_DIS
Enddeposition()
LIN {X 0.9725,Y -134.8573,Z 177,A -86.3065,B 6.5188,C 0.3905,E1 6.533,E2 538.3271} C_DIS
Startdeposition()
$VEL.CP = VEL_PRINT
LIN {X 2.4559,Y -135.7437,Z 177,A -84.3759,B 6.5379,C 0.3749,E1 6.557,E2 536.2561} C_DIS
LIN {X 8.6032,Y -135.4931,Z 177,A -82.8347,B 6.5371,C 0.39,E1 6.5609,E2 534.8499} C_DIS
LIN {X 15.0962,Y -134.925,Z 177,A -79.763,B 6.5374,C 0.3842,E1 6.5695,E2 531.7357} C_DIS
LIN {X 18.5236,Y -134.4978,Z 177,A -78.2903,B 6.5374,C 0.3832,E1 6.5736,E2 530.2602} C_DIS
LIN {X 23.1885,Y -133.7727,Z 177,A -76.3487,B 6.5374,C 0.3828,E1 6.579,E2 528.324} C_DIS
LIN {X 26.9642,Y -133.061,Z 177,A -74.8776,B 6.5374,C 0.384,E1 6.5829,E2 526.8712} C_DIS
LIN {X 29.5987,Y -132.5014,Z 177,A -73.6848,B 6.5375,C 0.3823,E1 6.5862,E2 525.6705} C_DIS
LIN {X 33.0696,Y -131.6768,Z 177,A -72.152,B 6.5376,C 0.3807,E1 6.5904,E2 524.1331} C_DIS
LIN {X 36.4409,Y -130.7835,Z 177,A -70.7362,B 6.5376,C 0.3803,E1 6.5942,E2 522.7235} C_DIS
LIN {X 39.789,Y -129.804,Z 177,A -69.2986,B 6.5376,C 0.3795,E1 6.598,E2 521.2893} C_DIS
LIN {X 45.4787,Y -127.9229,Z 177,A -66.8556,B 6.5377,C 0.3782,E1 6.6045,E2 518.8557} C_DIS
LIN {X 50.692,Y -125.9466,Z 177,A -64.2282,B 6.5381,C 0.3712,E1 6.6114,E2 516.1913} C_DIS
LIN {X 55.1789,Y -124.0466,Z 177,A -62.3527,B 6.5381,C 0.3715,E1 6.6162,E2 514.3375} C_DIS
LIN {X 58.1648,Y -122.6752,Z 177,A -60.9778,B 6.5382,C 0.3699,E1 6.6196,E2 512.9631} C_DIS
LIN {X 61.3268,Y -121.1251,Z 177,A -59.5599,B 6.5382,C 0.3689,E1 6.6232,E2 511.5527} C_DIS
LIN {X 64.7633,Y -119.3253,Z 177,A -57.8232,B 6.5385,C 0.3649,E1 6.6275,E2 509.802} C_DIS
LIN {X 68.6015,Y -117.1606,Z 177,A -55.9886,B 6.5386,C 0.3625,E1 6.6319,E2 507.9691} C_DIS
LIN {X 72.1453,Y -115.0128,Z 177,A -54.2854,B 6.5387,C 0.3605,E1 6.6359,E2 506.2704} C_DIS
LIN {X 75.4589,Y -112.8659,Z 177,A -52.6704,B 6.5389,C 0.3585,E1 6.6397,E2 504.6605} C_DIS
LIN {X 78.9331,Y -110.4641,Z 177,A -50.8889,B 6.539,C 0.3554,E1 6.6438,E2 502.8776} C_DIS
LIN {X 82.4015,Y -107.9015,Z 177,A -49.0779,B 6.5392,C 0.3523,E1 6.6478,E2 501.0662} C_DIS
LIN {X 85.7976,Y -105.2213,Z 177,A -47.2711,B 6.5394,C 0.3492,E1 6.6517,E2 499.2602} C_DIS
LIN {X 89.285,Y -102.2787,Z 177,A -45.4485,B 6.5394,C 0.3472,E1 6.6556,E2 497.4491} C_DIS
LIN {X 91.5935,Y -100.217,Z 177,A -43.6969,B 6.54,C 0.3371,E1 6.6593,E2 495.6391} C_DIS
LIN {X 94.7819,Y -97.2074,Z 177,A -42.2588,B 6.5398,C 0.3402,E1 6.6621,E2 494.2524} C_DIS
LIN {X 97.7275,Y -94.2451,Z 177,A -40.5269,B 6.54,C 0.337,E1 6.6655,E2 492.5228} C_DIS
LIN {X 100.8,Y -90.9518,Z 177,A -38.6578,B 6.5402,C 0.3334,E1 6.669,E2 490.6561} C_DIS
LIN {X 103.7419,Y -87.5816,Z 177,A -36.8039,B 6.5404,C 0.3297,E1 6.6724,E2 488.8048} C_DIS
LIN {X 106.4167,Y -84.3109,Z 177,A -35.115,B 6.5404,C 0.3272,E1 6.6753,E2 487.1263} C_DIS
LIN {X 108.9832,Y -80.9656,Z 177,A -33.3349,B 6.5407,C 0.3231,E1 6.6783,E2 485.3444} C_DIS
LIN {X 111.6391,Y -77.2629,Z 177,A -31.4209,B 6.5409,C 0.3186,E1 6.6814,E2 483.4298} C_DIS
LIN {X 114.124,Y -73.5433,Z 177,A -29.555,B 6.5411,C 0.3144,E1 6.6842,E2 481.5649} C_DIS
LIN {X 116.3984,Y -69.8881,Z 177,A -27.7527,B 6.5413,C 0.3101,E1 6.6869,E2 479.7627} C_DIS
LIN {X 118.6776,Y -65.9425,Z 177,A -26.1553,B 6.5413,C 0.3108,E1 6.689,E2 478.205} C_DIS
LIN {X 120.6679,Y -62.2249,Z 177,A -24.0841,B 6.5417,C 0.3012,E1 6.6918,E2 476.0949} C_DIS
LIN {X 122.4075,Y -58.7252,Z 177,A -22.6704,B 6.5417,C 0.301,E1 6.6934,E2 474.7097} C_DIS
LIN {X 123.6066,Y -56.1627,Z 177,A -21.3708,B 6.542,C 0.296,E1 6.695,E2 473.3957} C_DIS
LIN {X 124.9647,Y -53.0726,Z 177,A -20.0832,B 6.542,C 0.2946,E1 6.6964,E2 472.1242} C_DIS
LIN {X 126.871,Y -48.3379,Z 177,A -17.9914,B 6.5422,C 0.2899,E1 6.6985,E2 470.0382} C_DIS
LIN {X 128.7098,Y -43.1985,Z 177,A -15.6562,B 6.5425,C 0.283,E1 6.7007,E2 467.6969} C_DIS
LIN {X 129.7121,Y -40.0893,Z 177,A -14.4198,B 6.5425,C 0.2817,E1 6.7017,E2 466.4773} C_DIS
LIN {X 130.6689,Y -36.8507,Z 177,A -13.1625,B 6.5426,C 0.2807,E1 6.7027,E2 465.2398} C_DIS
LIN {X 132.1071,Y -31.3088,Z 177,A -10.5899,B 6.543,C 0.2712,E1 6.7045,E2 462.6455} C_DIS
LIN {X 132.9957,Y -27.2851,Z 177,A -9.0379,B 6.5431,C 0.2696,E1 6.7054,E2 461.1156} C_DIS
LIN {X 133.5239,Y -24.5785,Z 177,A -7.6867,B 6.5434,C 0.263,E1 6.7061,E2 459.7397} C_DIS
LIN {X 134.1218,Y -21.0647,Z 177,A -6.2533,B 6.5434,C 0.26,E1 6.7067,E2 458.3139} C_DIS
LIN {X 134.5961,Y -17.7824,Z 177,A -4.8476,B 6.5437,C 0.2559,E1 6.7072,E2 456.9062} C_DIS
LIN {X 135.0863,Y -13.5789,Z 177,A -3.1981,B 6.5437,C 0.2532,E1 6.7077,E2 455.2725} C_DIS
LIN {X 135.3646,Y -10.4442,Z 177,A -1.7853,B 6.544,C 0.2479,E1 6.7081,E2 453.8478} C_DIS
LIN {X 135.7166,Y -3.6552,Z 177,A 0.9718,B 6.5442,C 0.2416,E1 6.7084,E2 451.1024} C_DIS
LIN {X 135.764,Y 0.8635,Z 177,A 3.3273,B 6.5447,C 0.2283,E1 6.7084,E2 448.6887} C_DIS
LIN {X 135.66,Y 5.359,Z 177,A 5.1318,B 6.5447,C 0.2245,E1 6.7082,E2 446.8945} C_DIS
LIN {X 135.4239,Y 9.6311,Z 177,A 6.4752,B 6.5447,C 0.2274,E1 6.708,E2 445.6081} C_DIS
LIN {X 135.1009,Y 13.4268,Z 177,A 8.0816,B 6.5449,C 0.2229,E1 6.7075,E2 444.0007} C_DIS
LIN {X 134.6618,Y 17.2812,Z 177,A 9.6216,B 6.5449,C 0.2199,E1 6.707,E2 442.4717} C_DIS
LIN {X 134.1878,Y 20.6383,Z 177,A 11.0199,B 6.5451,C 0.2164,E1 6.7065,E2 441.0763} C_DIS
LIN {X 133.5733,Y 24.3027,Z 177,A 12.6431,B 6.5452,C 0.2111,E1 6.7057,E2 439.4451} C_DIS
LIN {X 132.76,Y 28.4096,Z 177,A 14.2971,B 6.5453,C 0.2081,E1 6.7047,E2 437.804} C_DIS
LIN {X 131.9977,Y 31.7627,Z 177,A 15.6563,B 6.5454,C 0.2056,E1 6.7039,E2 436.4553} C_DIS
LIN {X 131.2596,Y 34.6881,Z 177,A 16.9469,B 6.5455,C 0.2018,E1 6.703,E2 435.1617} C_DIS
LIN {X 130.351,Y 37.9591,Z 177,A 18.2091,B 6.5455,C 0.2008,E1 6.702,E2 433.9198} C_DIS
LIN {X 129.152,Y 41.8608,Z 177,A 20.1273,B 6.5458,C 0.1928,E1 6.7004,E2 431.9761} C_DIS
LIN {X 127.7922,Y 45.8414,Z 177,A 21.7541,B 6.5458,C 0.1905,E1 6.6989,E2 430.3667} C_DIS
LIN {X 126.5551,Y 49.1531,Z 177,A 23.8427,B 6.5463,C 0.1763,E1 6.6967,E2 428.2025} C_DIS
LIN {X 124.6303,Y 53.847,Z 177,A 25.3177,B 6.5461,C 0.1821,E1 6.6952,E2 426.8097} C_DIS
LIN {X 123.2529,Y 56.9291,Z 177,A 26.7268,B 6.5462,C 0.1786,E1 6.6936,E2 425.4019} C_DIS
LIN {X 121.9086,Y 59.7545,Z 177,A 27.9709,B 6.5462,C 0.1766,E1 6.6921,E2 424.1665} C_DIS
LIN {X 120.3649,Y 62.806,Z 177,A 29.4494,B 6.5464,C 0.1723,E1 6.6902,E2 422.6829} C_DIS
LIN {X 118.2503,Y 66.7057,Z 177,A 31.3573,B 6.5465,C 0.167,E1 6.6876,E2 420.7697} C_DIS
LIN {X 116.1124,Y 70.361,Z 177,A 33.135,B 6.5466,C 0.1628,E1 6.6851,E2 418.9924} C_DIS
LIN {X 113.6619,Y 74.2554,Z 177,A 34.967,B 6.5466,C 0.16,E1 6.6823,E2 417.1732} C_DIS
LIN {X 111.3197,Y 77.7221,Z 177,A 36.7506,B 6.5468,C 0.1555,E1 6.6795,E2 415.3866} C_DIS
LIN {X 108.6718,Y 81.3838,Z 177,A 38.6507,B 6.5468,C 0.1512,E1 6.6763,E2 413.4866} C_DIS
LIN {X 104.199,Y 87.0367,Z 177,A 41.6457,B 6.547,C 0.1453,E1 6.6711,E2 410.4965} C_DIS
LIN {X 101.1393,Y 90.5736,Z 177,A 43.5494,B 6.547,C 0.1422,E1 6.6676,E2 408.6009} C_DIS
LIN {X 96.6298,Y 95.3705,Z 177,A 46.2441,B 6.5472,C 0.1378,E1 6.6624,E2 405.9157} C_DIS
LIN {X 94.5826,Y 97.4008,Z 177,A 47.8636,B 6.5474,C 0.1288,E1 6.6591,E2 404.2462} C_DIS
LIN {X 91.4875,Y 100.314,Z 177,A 49.2774,B 6.5474,C 0.1315,E1 6.6563,E2 402.879} C_DIS
LIN {X 88.1671,Y 103.2443,Z 177,A 51.0891,B 6.5474,C 0.1289,E1 6.6525,E2 401.0741} C_DIS
LIN {X 84.8223,Y 106.0096,Z 177,A 52.9071,B 6.5474,C 0.1258,E1 6.6485,E2 399.2574} C_DIS
LIN {X 81.0766,Y 108.9005,Z 177,A 54.8537,B 6.5474,C 0.1232,E1 6.6442,E2 397.3168} C_DIS
LIN {X 77.519,Y 111.4609,Z 177,A 56.515,B 6.5474,C 0.1231,E1 6.6405,E2 395.6784} C_DIS
LIN {X 73.5006,Y 114.1514,Z 177,A 58.6539,B 6.5476,C 0.1183,E1 6.6355,E2 393.5273} C_DIS
LIN {X 69.9288,Y 116.3738,Z 177,A 60.4935,B 6.5476,C 0.1146,E1 6.6311,E2 391.6798} C_DIS
LIN {X 66.0389,Y 118.6242,Z 177,A 62.3731,B 6.5476,C 0.1122,E1 6.6265,E2 389.8023} C_DIS
LIN {X 61.9565,Y 120.8046,Z 177,A 64.2102,B 6.5476,C 0.1114,E1 6.622,E2 387.9794} C_DIS
LIN {X 58.8231,Y 122.3607,Z 177,A 65.5419,B 6.5476,C 0.1118,E1 6.6187,E2 386.6655} C_DIS
LIN {X 56.2461,Y 123.5687,Z 177,A 66.9831,B 6.5478,C 0.1066,E1 6.615,E2 385.1951} C_DIS
LIN {X 52.6223,Y 125.1527,Z 177,A 68.4625,B 6.5478,C 0.1076,E1 6.6112,E2 383.7389} C_DIS
LIN {X 49.7845,Y 126.3097,Z 177,A 69.8574,B 6.5478,C 0.1047,E1 6.6076,E2 382.3318} C_DIS
LIN {X 46.0874,Y 127.7035,Z 177,A 71.4157,B 6.5478,C 0.1047,E1 6.6035,E2 380.7871} C_DIS
LIN {X 42.9507,Y 128.7924,Z 177,A 72.813,B 6.5478,C 0.1034,E1 6.5998,E2 379.3905} C_DIS
LIN {X 35.8714,Y 130.9428,Z 177,A 76.0037,B 6.5478,C 0.0998,E1 6.5913,E2 376.1922} C_DIS
LIN {X 32.0774,Y 131.9219,Z 177,A 77.5977,B 6.5478,C 0.0995,E1 6.587,E2 374.6058} C_DIS
LIN {X 28.7044,Y 132.6964,Z 177,A 79.0353,B 6.5478,C 0.0989,E1 6.583,E2 373.1714} C_DIS
LIN {X 24.8353,Y 133.4764,Z 177,A 80.7822,B 6.5479,C 0.0968,E1 6.5782,E2 371.4152} C_DIS
LIN {X 20.8386,Y 134.1568,Z 177,A 82.2607,B 6.5479,C 0.0994,E1 6.5742,E2 369.9655} C_DIS
LIN {X 17.9982,Y 134.5678,Z 177,A 83.4176,B 6.5479,C 0.0997,E1 6.5711,E2 368.8156} C_DIS
LIN {X 14.3555,Y 135.0047,Z 177,A 85.558,B 6.548,C 0.0906,E1 6.5649,E2 366.6034} C_DIS
LIN {X 10.3703,Y 135.37,Z 177,A 86.8781,B 6.548,C 0.0955,E1 6.5614,E2 365.3291} C_DIS
LIN {X 6.122,Y 135.6294,Z 177,A 88.7954,B 6.548,C 0.0935,E1 6.556,E2 363.3978} C_DIS
LIN {X 1.173,Y 135.7614,Z 177,A 91.2058,B 6.548,C 0.0889,E1 6.5491,E2 360.949} C_DIS
LIN {X -3.2213,Y 135.7287,Z 177,A 92.6129,B 6.548,C 0.0952,E1 6.5454,E2 359.5975} C_DIS
LIN {X -6.9047,Y 135.5901,Z 177,A 94.152,B 6.548,C 0.0956,E1 6.5411,E2 358.0611} C_DIS
LIN {X -11.0823,Y 135.3131,Z 177,A 95.9355,B 6.548,C 0.0956,E1 6.5361,E2 356.2765} C_DIS
LIN {X -14.6783,Y 134.9699,Z 177,A 97.4516,B 6.548,C 0.0962,E1 6.5319,E2 354.7621} C_DIS
LIN {X -18.402,Y 134.5149,Z 177,A 99.1519,B 6.548,C 0.0952,E1 6.5272,E2 353.0485} C_DIS
LIN {X -22.1011,Y 133.9548,Z 177,A 100.6157,B 6.548,C 0.0974,E1 6.5232,E2 351.5996} C_DIS
LIN {X -25.4276,Y 133.3631,Z 177,A 101.973,B 6.5479,C 0.0991,E1 6.5194,E2 350.2514} C_DIS
LIN {X -28.6365,Y 132.711,Z 177,A 103.4481,B 6.5479,C 0.0986,E1 6.5154,E2 348.7659} C_DIS
LIN {X -32.7562,Y 131.7563,Z 177,A 105.2641,B 6.5479,C 0.0994,E1 6.5104,E2 346.9472} C_DIS
LIN {X -35.6029,Y 131.0156,Z 177,A 106.7784,B 6.5479,C 0.0967,E1 6.5063,E2 345.4004} C_DIS
LIN {X -38.9744,Y 130.0533,Z 177,A 107.9904,B 6.5479,C 0.1014,E1 6.5031,E2 344.2221} C_DIS
LIN {X -43.1051,Y 128.7409,Z 177,A 110.2156,B 6.5479,C 0.0978,E1 6.4971,E2 341.9497} C_DIS
LIN {X -46.9809,Y 127.3793,Z 177,A 111.8438,B 6.5479,C 0.1009,E1 6.4929,E2 340.3356} C_DIS
LIN {X -50.1332,Y 126.1718,Z 177,A 113.0828,B 6.5478,C 0.1048,E1 6.4897,E2 339.1204} C_DIS
LIN {X -53.9914,Y 124.5678,Z 177,A 114.7588,B 6.5478,C 0.1078,E1 6.4854,E2 337.4562} C_DIS
LIN {X -57.1291,Y 123.1604,Z 177,A 116.2167,B 6.5478,C 0.1095,E1 6.4817,E2 335.9985} C_DIS
LIN {X -60.3924,Y 121.5939,Z 177,A 117.8509,B 6.5478,C 0.11,E1 6.4776,E2 334.3525} C_DIS
LIN {X -64.8136,Y 119.2979,Z 177,A 119.9779,B 6.5477,C 0.1125,E1 6.4723,E2 332.2243} C_DIS
LIN {X -68.7261,Y 117.0875,Z 177,A 121.6351,B 6.5476,C 0.1182,E1 6.4684,E2 330.5976} C_DIS
LIN {X -74.8333,Y 113.2818,Z 177,A 124.9451,B 6.5476,C 0.1195,E1 6.4605,E2 327.257} C_DIS
LIN {X -78.4086,Y 110.8371,Z 177,A 126.8289,B 6.5476,C 0.1218,E1 6.4562,E2 325.368} C_DIS
LIN {X -82.0991,Y 108.1325,Z 177,A 128.7844,B 6.5474,C 0.1248,E1 6.4518,E2 323.4111} C_DIS
LIN {X -85.4641,Y 105.4928,Z 177,A 130.5857,B 6.5474,C 0.128,E1 6.4479,E2 321.6117} C_DIS
LIN {X -88.6763,Y 102.8069,Z 177,A 132.3509,B 6.5474,C 0.1313,E1 6.4441,E2 319.8482} C_DIS
LIN {X -91.8215,Y 100.0077,Z 177,A 134.1762,B 6.5473,C 0.1342,E1 6.4403,E2 318.0186} C_DIS
LIN {X -94.9893,Y 97.004,Z 177,A 136.0598,B 6.5472,C 0.1374,E1 6.4365,E2 316.1315} C_DIS
LIN {X -98.086,Y 93.8716,Z 177,A 137.9706,B 6.5472,C 0.1406,E1 6.4328,E2 314.2161} C_DIS
LIN {X -101.2531,Y 90.4465,Z 177,A 139.9611,B 6.547,C 0.1445,E1 6.4291,E2 312.2246} C_DIS
LIN {X -104.2518,Y 86.9738,Z 177,A 141.9575,B 6.547,C 0.148,E1 6.4255,E2 310.2227} C_DIS
LIN {X -107.1051,Y 83.4347,Z 177,A 143.9096,B 6.5469,C 0.152,E1 6.4221,E2 308.2682} C_DIS
LIN {X -109.8195,Y 79.8276,Z 177,A 145.8307,B 6.5468,C 0.1562,E1 6.4189,E2 306.3469} C_DIS
LIN {X -112.6911,Y 75.7207,Z 177,A 148.5759,B 6.5468,C 0.154,E1 6.4145,E2 303.526} C_DIS
LIN {X -115.5676,Y 71.2528,Z 177,A 149.9567,B 6.5465,C 0.1693,E1 6.4126,E2 302.2533} C_DIS
LIN {X -117.0894,Y 68.7228,Z 177,A 151.6504,B 6.5465,C 0.1673,E1 6.4101,E2 300.5059} C_DIS
LIN {X -119.2275,Y 64.9427,Z 177,A 154.031,B 6.5465,C 0.1657,E1 6.4068,E2 298.0593} C_DIS
LIN {X -121.7018,Y 60.1738,Z 177,A 155.5907,B 6.5462,C 0.1795,E1 6.405,E2 296.5891} C_DIS
LIN {X -123.0827,Y 57.2972,Z 177,A 157.2433,B 6.5462,C 0.1795,E1 6.403,E2 294.9001} C_DIS
LIN {X -125.1733,Y 52.573,Z 177,A 159.2138,B 6.546,C 0.1876,E1 6.4008,E2 292.9574} C_DIS
LIN {X -126.391,Y 49.5751,Z 177,A 160.712,B 6.5459,C 0.1898,E1 6.3993,E2 291.4441} C_DIS
LIN {X -128.0963,Y 44.9851,Z 177,A 162.9705,B 6.5458,C 0.1933,E1 6.3971,E2 289.1638} C_DIS
LIN {X -129.6749,Y 40.2109,Z 177,A 164.9295,B 6.5456,C 0.2009,E1 6.3954,E2 287.227} C_DIS
LIN {X -130.8173,Y 36.3199,Z 177,A 166.779,B 6.5455,C 0.2041,E1 6.394,E2 285.362} C_DIS
LIN {X -131.8856,Y 32.2279,Z 177,A 168.5358,B 6.5453,C 0.2094,E1 6.3928,E2 283.6102} C_DIS
LIN {X -132.7362,Y 28.5201,Z 177,A 170.1461,B 6.5452,C 0.2138,E1 6.3918,E2 282.0008} C_DIS
LIN {X -133.5557,Y 24.4006,Z 177,A 171.8827,B 6.545,C 0.2192,E1 6.3909,E2 280.2702} C_DIS
LIN {X -134.165,Y 20.7855,Z 177,A 173.5093,B 6.5449,C 0.2227,E1 6.3902,E2 278.635} C_DIS
LIN {X -134.6445,Y 17.4133,Z 177,A 175.0412,B 6.5448,C 0.2258,E1 6.3896,E2 277.0927} C_DIS
LIN {X -135.1222,Y 13.2047,Z 177,A 176.82,B 6.5446,C 0.2309,E1 6.3891,E2 275.3166} C_DIS
LIN {X -135.4195,Y 9.6918,Z 177,A 178.3894,B 6.5445,C 0.2343,E1 6.3888,E2 273.7382} C_DIS
LIN {X -135.6598,Y 5.3638,Z 177,A -179.7557,B 6.5443,C 0.2393,E1 6.3885,E2 271.8817} C_DIS
LIN {X -135.7625,Y 1.0843,Z 177,A -177.9954,B 6.5441,C 0.2449,E1 6.3885,E2 270.1287} C_DIS
LIN {X -135.7448,Y -2.3918,Z 177,A -176.401,B 6.544,C 0.2477,E1 6.3885,E2 268.5196} C_DIS
LIN {X -135.6007,Y -6.6937,Z 177,A -174.5377,B 6.5438,C 0.2524,E1 6.3887,E2 266.652} C_DIS
LIN {X -135.311,Y -11.1068,Z 177,A -172.6734,B 6.5436,C 0.2578,E1 6.3891,E2 264.7893} C_DIS
LIN {X -134.9832,Y -14.5555,Z 177,A -171.2318,B 6.5434,C 0.2621,E1 6.3895,E2 263.3515} C_DIS
LIN {X -134.5996,Y -17.7555,Z 177,A -169.805,B 6.5433,C 0.2652,E1 6.39,E2 261.9174} C_DIS
LIN {X -134.0377,Y -21.6042,Z 177,A -168.1241,B 6.5431,C 0.2694,E1 6.3907,E2 260.2328} C_DIS
LIN {X -133.3595,Y -25.4466,Z 177,A -166.4316,B 6.5429,C 0.2735,E1 6.3916,E2 258.5357} C_DIS
LIN {X -132.6373,Y -28.978,Z 177,A -164.8684,B 6.5428,C 0.2773,E1 6.3925,E2 256.9683} C_DIS
LIN {X -131.2634,Y -34.6738,Z 177,A -161.7081,B 6.5428,C 0.2764,E1 6.3947,E2 253.7232} C_DIS
LIN {X -129.8798,Y -39.5414,Z 177,A -160.0542,B 6.5423,C 0.2877,E1 6.396,E2 252.1314} C_DIS
LIN {X -128.5,Y -43.8231,Z 177,A -158.146,B 6.5421,C 0.2927,E1 6.3977,E2 250.2233} C_DIS
LIN {X -126.8283,Y -48.4504,Z 177,A -156.0147,B 6.5419,C 0.2976,E1 6.3997,E2 248.0864} C_DIS
LIN {X -125.418,Y -51.9872,Z 177,A -154.4404,B 6.5417,C 0.3021,E1 6.4014,E2 246.517} C_DIS
LIN {X -124.2167,Y -54.7987,Z 177,A -153.05,B 6.5416,C 0.3043,E1 6.403,E2 245.1149} C_DIS
LIN {X -122.1542,Y -59.255,Z 177,A -150.8886,B 6.5414,C 0.3086,E1 6.4055,E2 242.9434} C_DIS
LIN {X -120.4054,Y -62.729,Z 177,A -149.4761,B 6.5411,C 0.3154,E1 6.4073,E2 241.5604} C_DIS
LIN {X -117.2071,Y -68.5223,Z 177,A -146.391,B 6.5409,C 0.3188,E1 6.4116,E2 238.44} C_DIS
LIN {X -114.9094,Y -72.3091,Z 177,A -144.5381,B 6.5407,C 0.3235,E1 6.4143,E2 236.59} C_DIS
LIN {X -110.9051,Y -78.3123,Z 177,A -141.6051,B 6.5403,C 0.3319,E1 6.4189,E2 233.6726} C_DIS
LIN {X -107.0164,Y -83.5488,Z 177,A -138.5764,B 6.5401,C 0.3348,E1 6.424,E2 230.6101} C_DIS
LIN {X -104.1486,Y -87.0969,Z 177,A -136.6336,B 6.5399,C 0.3387,E1 6.4275,E2 228.6658} C_DIS
LIN {X -101.6878,Y -89.9574,Z 177,A -135.1806,B 6.5396,C 0.3437,E1 6.4301,E2 227.2309} C_DIS
LIN {X -98.7149,Y -93.21,Z 177,A -133.1796,B 6.5396,C 0.3458,E1 6.4339,E2 225.2126} C_DIS
LIN {X -95.5868,Y -96.4154,Z 177,A -131.2525,B 6.5394,C 0.349,E1 6.4377,E2 223.2812} C_DIS
LIN {X -92.3429,Y -99.5268,Z 177,A -129.3037,B 6.5392,C 0.352,E1 6.4417,E2 221.3263} C_DIS
LIN {X -88.9702,Y -102.5533,Z 177,A -127.3233,B 6.5391,C 0.3546,E1 6.4459,E2 219.3377} C_DIS
LIN {X -86.531,Y -104.619,Z 177,A -125.8823,B 6.5391,C 0.3558,E1 6.449,E2 217.8851} C_DIS
LIN {X -82.5802,Y -107.7648,Z 177,A -123.8413,B 6.5387,C 0.3605,E1 6.4534,E2 215.856} C_DIS
LIN {X -77.068,Y -111.7737,Z 177,A -120.9066,B 6.5385,C 0.3643,E1 6.4601,E2 212.9141} C_DIS
LIN {X -73.6152,Y -114.0775,Z 177,A -119.1103,B 6.5385,C 0.3663,E1 6.4643,E2 211.1123} C_DIS
LIN {X -69.7058,Y -116.5071,Z 177,A -117.1697,B 6.5383,C 0.369,E1 6.469,E2 209.172} C_DIS
LIN {X -65.6985,Y -118.8127,Z 177,A -115.2176,B 6.5381,C 0.3716,E1 6.4737,E2 207.2198} C_DIS
LIN {X -61.8668,Y -120.8503,Z 177,A -113.6103,B 6.5378,C 0.3768,E1 6.4776,E2 205.6409} C_DIS
LIN {X -59.2441,Y -122.1596,Z 177,A -112.2165,B 6.5378,C 0.3761,E1 6.4812,E2 204.2271} C_DIS
LIN {X -56.1253,Y -123.6233,Z 177,A -110.7454,B 6.5378,C 0.3775,E1 6.4849,E2 202.7538} C_DIS
LIN {X -52.6565,Y -125.1384,Z 177,A -109.0243,B 6.5378,C 0.3775,E1 6.4894,E2 201.0165} C_DIS
LIN {X -48.7692,Y -126.7043,Z 177,A -107.2105,B 6.5378,C 0.3785,E1 6.4941,E2 199.1968} C_DIS
LIN {X -43.7581,Y -128.5225,Z 177,A -104.4808,B 6.538,C 0.3738,E1 6.5015,E2 196.405} C_DIS
LIN {X -39.0724,Y -130.0233,Z 177,A -102.9027,B 6.5375,C 0.3822,E1 6.5055,E2 194.8906} C_DIS
LIN {X -35.5417,Y -131.032,Z 177,A -101.3784,B 6.5375,C 0.3836,E1 6.5096,E2 193.3692} C_DIS
LIN {X -31.9921,Y -131.9424,Z 177,A -99.9219,B 6.5373,C 0.3857,E1 6.5135,E2 191.9238} C_DIS
LIN {X -29.0427,Y -132.6234,Z 177,A -98.5715,B 6.5373,C 0.3853,E1 6.5172,E2 190.5637} C_DIS
LIN {X -25.5714,Y -133.3356,Z 177,A -97.1066,B 6.5373,C 0.3864,E1 6.5212,E2 189.1022} C_DIS
LIN {X -22.2408,Y -133.9315,Z 177,A -95.689,B 6.5373,C 0.3871,E1 6.5251,E2 187.6855} C_DIS
LIN {X -19.2138,Y -134.3991,Z 177,A -94.2935,B 6.5373,C 0.386,E1 6.529,E2 186.2763} C_DIS
LIN {X -13.0966,Y -135.1326,Z 177,A -91.7316,B 6.5373,C 0.3871,E1 6.5361,E2 183.7184} C_DIS
LIN {X -10.0335,Y -135.3945,Z 177,A -90.1129,B 6.5375,C 0.3825,E1 6.5408,E2 182.0579} C_DIS
LIN {X -6.3357,Y -135.6187,Z 177,A -88.9622,B 6.5371,C 0.3886,E1 6.5438,E2 180.9596} C_DIS
LIN {X 0.6203,Y -135.7645,Z 177,A -85.9546,B 6.5372,C 0.3873,E1 6.5523,E2 177.9417} C_DIS
LIN {X 0.6203,Y -135.7645,Z 177,A -85.9546,B 6.5372,C 0.3873,E1 6.5523,E2 177.9417} C_DIS
Enddeposition()
LIN {X 0.9877,Y -136.6672,Z 177,A -86.2019,B 6.5407,C 0.397,E1 6.5554,E2 178.2721} C_DIS
Startdeposition()
$VEL.CP = VEL_PRINT
LIN {X -3.0776,Y -136.6378,Z 177,A -88.2948,B 6.5404,C 0.4028,E1 6.5494,E2 180.4156} C_DIS
LIN {X -7.1982,Y -136.4813,Z 177,A -90.3874,B 6.5401,C 0.408,E1 6.5435,E2 182.5552} C_DIS
LIN {X -11.6786,Y -136.1707,Z 177,A -91.6895,B 6.5406,C 0.3995,E1 6.54,E2 183.7842} C_DIS
LIN {X -18.7279,Y -135.3825,Z 177,A -95.1962,B 6.5402,C 0.4064,E1 6.5301,E2 187.3599} C_DIS
LIN {X -22.8311,Y -134.7503,Z 177,A -96.4873,B 6.5406,C 0.3995,E1 6.5267,E2 188.5944} C_DIS
LIN {X -26.9179,Y -133.9937,Z 177,A -98.2595,B 6.5406,C 0.3991,E1 6.5218,E2 190.3709} C_DIS
LIN {X -30.5787,Y -133.2056,Z 177,A -99.8065,B 6.5406,C 0.398,E1 6.5176,E2 191.9154} C_DIS
LIN {X -33.741,Y -132.4398,Z 177,A -101.1751,B 6.5407,C 0.3973,E1 6.5139,E2 193.285} C_DIS
LIN {X -37.1928,Y -131.5127,Z 177,A -102.6902,B 6.5407,C 0.3966,E1 6.5098,E2 194.8026} C_DIS
LIN {X -40.9648,Y -130.3881,Z 177,A -104.553,B 6.5407,C 0.3983,E1 6.5048,E2 196.6928} C_DIS
LIN {X -45.6397,Y -128.8267,Z 177,A -106.3775,B 6.541,C 0.3933,E1 6.5,E2 198.4869} C_DIS
LIN {X -48.2143,Y -127.8835,Z 177,A -107.5716,B 6.541,C 0.3929,E1 6.4969,E2 199.6868} C_DIS
LIN {X -51.761,Y -126.4912,Z 177,A -109.1666,B 6.541,C 0.3914,E1 6.4928,E2 201.2818} C_DIS
LIN {X -54.4088,Y -125.3731,Z 177,A -110.4164,B 6.5411,C 0.3907,E1 6.4895,E2 202.5373} C_DIS
LIN {X -57.6821,Y -123.9015,Z 177,A -111.9191,B 6.5412,C 0.3891,E1 6.4857,E2 204.0399} C_DIS
LIN {X -61.0738,Y -122.2667,Z 177,A -113.5011,B 6.5413,C 0.3873,E1 6.4818,E2 205.6226} C_DIS
LIN {X -64.3395,Y -120.5812,Z 177,A -115.1845,B 6.5413,C 0.3873,E1 6.4776,E2 207.3242} C_DIS
LIN {X -68.2675,Y -118.4012,Z 177,A -117.0451,B 6.5415,C 0.3845,E1 6.473,E2 209.1819} C_DIS
LIN {X -71.9491,Y -116.201,Z 177,A -118.8806,B 6.5415,C 0.3825,E1 6.4686,E2 211.022} C_DIS
LIN {X -75.5998,Y -113.8597,Z 177,A -120.7161,B 6.5417,C 0.38,E1 6.4643,E2 212.8597} C_DIS
LIN {X -79.4992,Y -111.1716,Z 177,A -122.7248,B 6.5419,C 0.3772,E1 6.4597,E2 214.8711} C_DIS
LIN {X -83.051,Y -108.5439,Z 177,A -124.5909,B 6.5421,C 0.3744,E1 6.4556,E2 216.7388} C_DIS
LIN {X -86.5758,Y -105.7539,Z 177,A -126.52,B 6.5422,C 0.3717,E1 6.4514,E2 218.6732} C_DIS
LIN {X -90.1044,Y -102.7645,Z 177,A -128.4791,B 6.5424,C 0.3685,E1 6.4472,E2 220.6346} C_DIS
LIN {X -93.3102,Y -99.8624,Z 177,A -130.3066,B 6.5426,C 0.3653,E1 6.4435,E2 222.4635} C_DIS
LIN {X -96.4499,Y -96.8332,Z 177,A -132.1715,B 6.5427,C 0.3622,E1 6.4397,E2 224.3325} C_DIS
LIN {X -99.6164,Y -93.5722,Z 177,A -134.5065,B 6.5427,C 0.3636,E1 6.4351,E2 226.7209} C_DIS
LIN {X -102.5279,Y -90.3731,Z 177,A -135.9159,B 6.5431,C 0.355,E1 6.4326,E2 228.079} C_DIS
LIN {X -105.3824,Y -87.0277,Z 177,A -137.8177,B 6.5433,C 0.3517,E1 6.4292,E2 229.9876} C_DIS
LIN {X -108.2262,Y -83.4652,Z 177,A -139.9127,B 6.5434,C 0.3497,E1 6.4255,E2 232.105} C_DIS
LIN {X -110.8098,Y -80.003,Z 177,A -141.6076,B 6.5437,C 0.3443,E1 6.4228,E2 233.7847} C_DIS
LIN {X -113.2494,Y -76.5103,Z 177,A -143.5541,B 6.5438,C 0.342,E1 6.4197,E2 235.7505} C_DIS
LIN {X -115.8259,Y -72.5518,Z 177,A -145.4619,B 6.5441,C 0.3365,E1 6.4168,E2 237.6484} C_DIS
LIN {X -118.1302,Y -68.7357,Z 177,A -147.5091,B 6.5442,C 0.3341,E1 6.4139,E2 239.7171} C_DIS
LIN {X -120.091,Y -65.2492,Z 177,A -149.0715,B 6.5445,C 0.3286,E1 6.4118,E2 241.2644} C_DIS
LIN {X -121.9123,Y -61.775,Z 177,A -150.6537,B 6.5448,C 0.3238,E1 6.4098,E2 242.8378} C_DIS
LIN {X -123.544,Y -58.4451,Z 177,A -152.2309,B 6.5449,C 0.3201,E1 6.4079,E2 244.4171} C_DIS
LIN {X -124.8368,Y -55.6282,Z 177,A -153.5566,B 6.5451,C 0.317,E1 6.4063,E2 245.7454} C_DIS
LIN {X -126.1124,Y -52.6722,Z 177,A -154.9838,B 6.5452,C 0.3144,E1 6.4048,E2 247.1814} C_DIS
LIN {X -127.531,Y -49.1399,Z 177,A -156.6016,B 6.5454,C 0.3104,E1 6.4031,E2 248.8011} C_DIS
LIN {X -129.8262,Y -42.7097,Z 177,A -159.5707,B 6.5457,C 0.304,E1 6.4004,E2 251.7817} C_DIS
LIN {X -132.411,Y -33.8548,Z 177,A -163.4591,B 6.5462,C 0.2937,E1 6.3974,E2 255.6704} C_DIS
LIN {X -133.1124,Y -30.9867,Z 177,A -164.7887,B 6.5462,C 0.2913,E1 6.3965,E2 257.0106} C_DIS
LIN {X -133.9579,Y -27.094,Z 177,A -166.3595,B 6.5465,C 0.2855,E1 6.3956,E2 258.5678} C_DIS
LIN {X -134.5762,Y -23.8345,Z 177,A -167.7919,B 6.5467,C 0.2821,E1 6.3949,E2 260.0044} C_DIS
LIN {X -135.1565,Y -20.2955,Z 177,A -169.5103,B 6.5467,C 0.2802,E1 6.3941,E2 261.7484} C_DIS
LIN {X -135.7053,Y -16.2134,Z 177,A -171.1547,B 6.547,C 0.2744,E1 6.3936,E2 263.3813} C_DIS
LIN {X -136.1164,Y -12.3164,Z 177,A -172.9686,B 6.5471,C 0.2716,E1 6.3931,E2 265.2152} C_DIS
LIN {X -136.4275,Y -8.1501,Z 177,A -174.67,B 6.5473,C 0.2661,E1 6.3928,E2 266.909} C_DIS
LIN {X -136.6223,Y -3.6359,Z 177,A -176.546,B 6.5476,C 0.2605,E1 6.3926,E2 268.7812} C_DIS
LIN {X -136.6727,Y 0.2944,Z 177,A -178.3655,B 6.5476,C 0.2576,E1 6.3926,E2 270.6207} C_DIS
LIN {X -136.601,Y 4.4004,Z 177,A 179.8743,B 6.5479,C 0.2531,E1 6.3926,E2 272.3842} C_DIS
LIN {X -136.4108,Y 8.4217,Z 177,A 178.2466,B 6.5481,C 0.2476,E1 6.3929,E2 274.003} C_DIS
LIN {X -136.117,Y 12.3106,Z 177,A 176.4443,B 6.5481,C 0.2448,E1 6.3933,E2 275.8246} C_DIS
LIN {X -135.6865,Y 16.3712,Z 177,A 174.8521,B 6.5484,C 0.2386,E1 6.3938,E2 277.4006} C_DIS
LIN {X -135.176,Y 20.1692,Z 177,A 173.0852,B 6.5484,C 0.2358,E1 6.3945,E2 279.1859} C_DIS
LIN {X -134.5052,Y 24.2311,Z 177,A 171.4836,B 6.5487,C 0.2296,E1 6.3953,E2 280.7706} C_DIS
LIN {X -133.9037,Y 27.36,Z 177,A 170.0977,B 6.5488,C 0.2263,E1 6.396,E2 282.1615} C_DIS
LIN {X -133.186,Y 30.6643,Z 177,A 168.5955,B 6.5489,C 0.2233,E1 6.397,E2 283.6729} C_DIS
LIN {X -132.225,Y 34.5794,Z 177,A 166.8159,B 6.5491,C 0.2196,E1 6.3982,E2 285.4619} C_DIS
LIN {X -130.4234,Y 40.8541,Z 177,A 163.0716,B 6.5489,C 0.223,E1 6.4013,E2 289.3262} C_DIS
LIN {X -128.1413,Y 47.5259,Z 177,A 161.2429,B 6.5496,C 0.2027,E1 6.4029,E2 291.0151} C_DIS
LIN {X -126.6242,Y 51.4311,Z 177,A 159.2794,B 6.5496,C 0.2003,E1 6.405,E2 293.0024} C_DIS
LIN {X -125.2069,Y 54.7933,Z 177,A 157.7172,B 6.5498,C 0.1966,E1 6.4067,E2 294.5673} C_DIS
LIN {X -123.8733,Y 57.7431,Z 177,A 156.3084,B 6.5498,C 0.1937,E1 6.4083,E2 295.9811} C_DIS
LIN {X -122.3489,Y 60.9072,Z 177,A 154.4814,B 6.5498,C 0.1938,E1 6.4106,E2 297.8499} C_DIS
LIN {X -120.6775,Y 64.1569,Z 177,A 153.4247,B 6.5501,C 0.1846,E1 6.4119,E2 298.8473} C_DIS
LIN {X -119.0279,Y 67.1689,Z 177,A 151.7355,B 6.5501,C 0.1838,E1 6.4143,E2 300.5658} C_DIS
LIN {X -116.8372,Y 70.9109,Z 177,A 149.6549,B 6.5501,C 0.1823,E1 6.4173,E2 302.6766} C_DIS
LIN {X -115.1084,Y 73.6837,Z 177,A 148.3402,B 6.5503,C 0.1783,E1 6.4192,E2 303.9834} C_DIS
LIN {X -112.3761,Y 77.7879,Z 177,A 146.3306,B 6.5505,C 0.1728,E1 6.4224,E2 305.9841} C_DIS
LIN {X -109.7144,Y 81.4986,Z 177,A 144.4173,B 6.5505,C 0.1683,E1 6.4255,E2 307.8955} C_DIS
LIN {X -107.1493,Y 84.8432,Z 177,A 142.5736,B 6.5506,C 0.1652,E1 6.4287,E2 309.7469} C_DIS
LIN {X -104.2377,Y 88.3955,Z 177,A 140.6527,B 6.5508,C 0.1609,E1 6.4321,E2 311.6655} C_DIS
LIN {X -101.3538,Y 91.6879,Z 177,A 138.7648,B 6.5508,C 0.1576,E1 6.4357,E2 313.5582} C_DIS
LIN {X -98.2037,Y 95.0541,Z 177,A 136.828,B 6.5509,C 0.1536,E1 6.4394,E2 315.4938} C_DIS
LIN {X -95.0524,Y 98.2052,Z 177,A 134.9334,B 6.551,C 0.1502,E1 6.4431,E2 317.3899} C_DIS
LIN {X -91.6995,Y 101.3433,Z 177,A 132.9764,B 6.551,C 0.1468,E1 6.4472,E2 319.349} C_DIS
LIN {X -88.2823,Y 104.3339,Z 177,A 131.0252,B 6.5511,C 0.1438,E1 6.4513,E2 321.3044} C_DIS
LIN {X -84.7597,Y 107.2157,Z 177,A 129.0817,B 6.5512,C 0.1408,E1 6.4555,E2 323.2506} C_DIS
LIN {X -81.2519,Y 109.8978,Z 177,A 127.1915,B 6.5512,C 0.1381,E1 6.4598,E2 325.1439} C_DIS
LIN {X -77.5895,Y 112.5132,Z 177,A 125.3147,B 6.5513,C 0.1349,E1 6.4641,E2 327.018} C_DIS
LIN {X -74.0003,Y 114.9058,Z 177,A 123.2509,B 6.5513,C 0.1352,E1 6.469,E2 329.1111} C_DIS
LIN {X -71.0956,Y 116.7255,Z 177,A 121.9875,B 6.5514,C 0.1309,E1 6.4719,E2 330.3525} C_DIS
LIN {X -67.2498,Y 118.9824,Z 177,A 120.1087,B 6.5514,C 0.1284,E1 6.4765,E2 332.2309} C_DIS
LIN {X -63.5051,Y 121.0198,Z 177,A 118.4446,B 6.5515,C 0.1244,E1 6.4805,E2 333.8787} C_DIS
LIN {X -59.8932,Y 122.8491,Z 177,A 116.7333,B 6.5515,C 0.1225,E1 6.4848,E2 335.5904} C_DIS
LIN {X -56.9882,Y 124.2224,Z 177,A 115.3187,B 6.5515,C 0.1217,E1 6.4884,E2 337.0122} C_DIS
LIN {X -53.1193,Y 125.9257,Z 177,A 113.26,B 6.5515,C 0.1233,E1 6.4938,E2 339.1042} C_DIS
LIN {X -50.0383,Y 127.1817,Z 177,A 112.2665,B 6.5517,C 0.1168,E1 6.4962,E2 340.0483} C_DIS
LIN {X -43.6852,Y 129.5014,Z 177,A 109.4188,B 6.5517,C 0.1142,E1 6.5037,E2 342.8956} C_DIS
LIN {X -39.639,Y 130.7961,Z 177,A 107.4161,B 6.5517,C 0.1156,E1 6.5091,E2 344.924} C_DIS
LIN {X -35.1244,Y 132.0796,Z 177,A 105.5068,B 6.5517,C 0.1134,E1 6.5142,E2 346.825} C_DIS
LIN {X -31.7795,Y 132.9244,Z 177,A 104.0372,B 6.5517,C 0.1127,E1 6.5182,E2 348.2964} C_DIS
LIN {X -27.7141,Y 133.8317,Z 177,A 102.2657,B 6.5517,C 0.112,E1 6.523,E2 350.07} C_DIS
LIN {X -23.9927,Y 134.5479,Z 177,A 100.7598,B 6.5517,C 0.1101,E1 6.5271,E2 351.5649} C_DIS
LIN {X -20.8609,Y 135.0689,Z 177,A 99.3858,B 6.5517,C 0.1101,E1 6.5309,E2 352.9433} C_DIS
LIN {X -17.4659,Y 135.5501,Z 177,A 97.9081,B 6.5517,C 0.1101,E1 6.5351,E2 354.4251} C_DIS
LIN {X -13.3918,Y 136.0132,Z 177,A 96.1641,B 6.5518,C 0.1099,E1 6.5399,E2 356.1713} C_DIS
LIN {X -9.69,Y 136.3268,Z 177,A 94.367,B 6.5518,C 0.1129,E1 6.545,E2 357.9966} C_DIS
LIN {X -6.3518,Y 136.5238,Z 177,A 93.3559,B 6.5518,C 0.1074,E1 6.5477,E2 358.9597} C_DIS
LIN {X 2.1237,Y 136.6542,Z 177,A 89.9047,B 6.5518,C 0.1059,E1 6.5573,E2 362.3969} C_DIS
LIN {X 7.7792,Y 136.4504,Z 177,A 87.4195,B 6.5518,C 0.1078,E1 6.5643,E2 364.895} C_DIS
LIN {X 11.8802,Y 136.1537,Z 177,A 84.6891,B 6.5516,C 0.1224,E1 6.5722,E2 367.7459} C_DIS
Enddeposition()
END
